ABB RAPID module: MainModule.mod

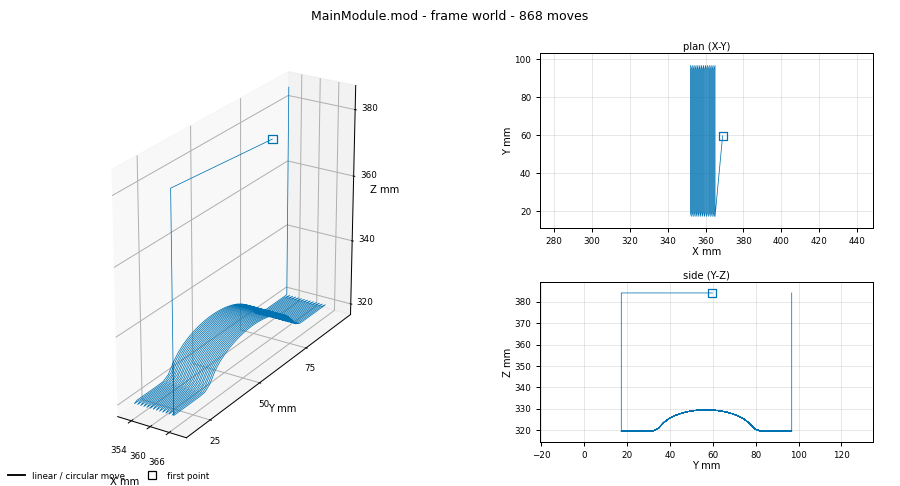
[picture p0: tool path of MainModule.mod in frame world, 868 of 868 moves have a stored position in this frame; points joined in program order, loops and branches not executed]
MODULE MainModule
PERS wobjdata Workobject_1:=[FALSE,TRUE,"",[[349,99.8,314.1],[0.707106781,0,0,-0.707106781]],[[0,0,0],[1,0,0,0]]];
PERS tooldata Extruder:=[TRUE,[[-32.5,-6.5,85.6],[0,-0.707106781,0.707106781,0]],[0.5,[-3,-15,42],[1,0,0,0],0,0,0]];
CONST robtarget p1 := [ [0,0,0], [1, 0, 0, 0], [0,0,0,0], [9E9,9E9, 9E9, 9E9, 9E9, 9E9] ];
VAR speeddata vel1 := [20,20,10,10];
VAR zonedata zoneval:=[FALSE,5,30,30,10,10,10];



PROC main()
AccSet 10,10;
SingArea\Wrist;
ConfL\On;

MoveL RelTool (p1,40.000000,20.000000,70.00000,\Rx:=0.000000,\Ry:=0.000000),vel1,z0,Extruder\WObj:=Workobject_1;
MoveL RelTool (p1,82.500000,16.000000,70.00000,\Rx:=0.000000,\Ry:=0.000000),vel1,z0,Extruder\WObj:=Workobject_1;


MoveL RelTool (p1,82.500000,16.000000,5.500000,\Rx:=0.000000,\Ry:=-0.000000),vel1,zoneval,Extruder\WObj:=Workobject_1;
MoveL RelTool (p1,80.000000,16.000000,5.500000,\Rx:=0.000000,\Ry:=-0.000000),vel1,zoneval,Extruder\WObj:=Workobject_1;
MoveL RelTool (p1,77.500000,16.000000,5.500000,\Rx:=0.000000,\Ry:=-0.000000),vel1,zoneval,Extruder\WObj:=Workobject_1;
MoveL RelTool (p1,75.000000,16.000000,5.500000,\Rx:=0.000000,\Ry:=-0.000000),vel1,zoneval,Extruder\WObj:=Workobject_1;
MoveL RelTool (p1,72.500000,16.000000,5.500000,\Rx:=0.000000,\Ry:=-0.000000),vel1,zoneval,Extruder\WObj:=Workobject_1;
MoveL RelTool (p1,70.000000,16.000000,5.500000,\Rx:=0.000000,\Ry:=-0.000000),vel1,zoneval,Extruder\WObj:=Workobject_1;
MoveL RelTool (p1,67.500000,16.000000,5.696103,\Rx:=0.000000,\Ry:=2.996421),vel1,zoneval,Extruder\WObj:=Workobject_1;
MoveL RelTool (p1,65.000000,16.000000,7.002928,\Rx:=0.000000,\Ry:=8.615508),vel1,zoneval,Extruder\WObj:=Workobject_1;
MoveL RelTool (p1,62.500000,16.000000,9.740509,\Rx:=0.000000,\Ry:=9.749555),vel1,zoneval,Extruder\WObj:=Workobject_1;
MoveL RelTool (p1,60.000000,16.000000,11.535030,\Rx:=0.000000,\Ry:=7.277441),vel1,zoneval,Extruder\WObj:=Workobject_1;
MoveL RelTool (p1,57.500000,16.000000,12.769306,\Rx:=0.000000,\Ry:=4.894735),vel1,zoneval,Extruder\WObj:=Workobject_1;
MoveL RelTool (p1,55.000000,16.000000,13.693467,\Rx:=0.000000,\Ry:=3.765598),vel1,zoneval,Extruder\WObj:=Workobject_1;
MoveL RelTool (p1,52.500000,16.000000,14.391107,\Rx:=0.000000,\Ry:=2.777529),vel1,zoneval,Extruder\WObj:=Workobject_1;
MoveL RelTool (p1,50.000000,16.000000,14.902666,\Rx:=0.000000,\Ry:=1.838961),vel1,zoneval,Extruder\WObj:=Workobject_1;
MoveL RelTool (p1,47.500000,16.000000,15.253646,\Rx:=0.000000,\Ry:=1.522915),vel1,zoneval,Extruder\WObj:=Workobject_1;
MoveL RelTool (p1,45.000000,16.000000,15.441995,\Rx:=0.000000,\Ry:=0.957446),vel1,zoneval,Extruder\WObj:=Workobject_1;
MoveL RelTool (p1,42.500000,16.000000,15.493202,\Rx:=0.000000,\Ry:=0.175753),vel1,zoneval,Extruder\WObj:=Workobject_1;
MoveL RelTool (p1,40.000000,16.000000,15.385044,\Rx:=0.000000,\Ry:=-0.609665),vel1,zoneval,Extruder\WObj:=Workobject_1;
MoveL RelTool (p1,37.500000,16.000000,15.140411,\Rx:=0.000000,\Ry:=-1.473255),vel1,zoneval,Extruder\WObj:=Workobject_1;
MoveL RelTool (p1,35.000000,16.000000,14.745289,\Rx:=0.000000,\Ry:=-2.361471),vel1,zoneval,Extruder\WObj:=Workobject_1;
MoveL RelTool (p1,32.500000,16.000000,14.177969,\Rx:=0.000000,\Ry:=-3.310711),vel1,zoneval,Extruder\WObj:=Workobject_1;
MoveL RelTool (p1,30.000000,16.000000,13.409588,\Rx:=0.000000,\Ry:=-4.304408),vel1,zoneval,Extruder\WObj:=Workobject_1;
MoveL RelTool (p1,27.500000,16.000000,12.393895,\Rx:=0.000000,\Ry:=-5.366573),vel1,zoneval,Extruder\WObj:=Workobject_1;
MoveL RelTool (p1,25.000000,16.000000,11.015814,\Rx:=0.000000,\Ry:=-7.116071),vel1,zoneval,Extruder\WObj:=Workobject_1;
MoveL RelTool (p1,22.500000,16.000000,8.916208,\Rx:=0.000000,\Ry:=-10.083054),vel1,zoneval,Extruder\WObj:=Workobject_1;
MoveL RelTool (p1,20.000000,16.000000,6.390765,\Rx:=0.000000,\Ry:=-7.195088),vel1,zoneval,Extruder\WObj:=Workobject_1;
MoveL RelTool (p1,17.500000,16.000000,5.549338,\Rx:=0.000000,\Ry:=-1.638714),vel1,zoneval,Extruder\WObj:=Workobject_1;
MoveL RelTool (p1,15.000000,16.000000,5.500000,\Rx:=0.000000,\Ry:=-0.000000),vel1,zoneval,Extruder\WObj:=Workobject_1;
MoveL RelTool (p1,12.500000,16.000000,5.500000,\Rx:=0.000000,\Ry:=-0.000000),vel1,zoneval,Extruder\WObj:=Workobject_1;
MoveL RelTool (p1,10.000000,16.000000,5.500000,\Rx:=0.000000,\Ry:=-0.000000),vel1,zoneval,Extruder\WObj:=Workobject_1;
MoveL RelTool (p1,7.500000,16.000000,5.500000,\Rx:=0.000000,\Ry:=-0.000000),vel1,zoneval,Extruder\WObj:=Workobject_1;
MoveL RelTool (p1,5.000000,16.000000,5.500000,\Rx:=0.000000,\Ry:=-0.000000),vel1,zoneval,Extruder\WObj:=Workobject_1;
MoveL RelTool (p1,3.000000,16.000000,5.500000,\Rx:=0.000000,\Ry:=0),vel1,zoneval,Extruder\WObj:=Workobject_1;
MoveL RelTool (p1,5.000000,15.500000,5.500000,\Rx:=0.000000,\Ry:=0.000000),vel1,zoneval,Extruder\WObj:=Workobject_1;
MoveL RelTool (p1,7.500000,15.500000,5.500000,\Rx:=0.000000,\Ry:=0.000000),vel1,zoneval,Extruder\WObj:=Workobject_1;
MoveL RelTool (p1,10.000000,15.500000,5.500000,\Rx:=0.000000,\Ry:=0.000000),vel1,zoneval,Extruder\WObj:=Workobject_1;
MoveL RelTool (p1,12.500000,15.500000,5.500000,\Rx:=0.000000,\Ry:=0.000000),vel1,zoneval,Extruder\WObj:=Workobject_1;
MoveL RelTool (p1,15.000000,15.500000,5.500000,\Rx:=0.000000,\Ry:=0.000000),vel1,zoneval,Extruder\WObj:=Workobject_1;
MoveL RelTool (p1,17.500000,15.500000,5.549338,\Rx:=0.000000,\Ry:=-1.027233),vel1,zoneval,Extruder\WObj:=Workobject_1;
MoveL RelTool (p1,20.000000,15.500000,6.390765,\Rx:=0.000000,\Ry:=-6.482955),vel1,zoneval,Extruder\WObj:=Workobject_1;
MoveL RelTool (p1,22.500000,15.500000,8.916208,\Rx:=0.000000,\Ry:=-11.282192),vel1,zoneval,Extruder\WObj:=Workobject_1;
MoveL RelTool (p1,25.000000,15.500000,11.015814,\Rx:=0.000000,\Ry:=-7.926142),vel1,zoneval,Extruder\WObj:=Workobject_1;
MoveL RelTool (p1,27.500000,15.500000,12.393895,\Rx:=0.000000,\Ry:=-5.366573),vel1,zoneval,Extruder\WObj:=Workobject_1;
MoveL RelTool (p1,30.000000,15.500000,13.409588,\Rx:=0.000000,\Ry:=-4.304408),vel1,zoneval,Extruder\WObj:=Workobject_1;
MoveL RelTool (p1,32.500000,15.500000,14.177969,\Rx:=0.000000,\Ry:=-3.310711),vel1,zoneval,Extruder\WObj:=Workobject_1;
MoveL RelTool (p1,35.000000,15.500000,14.745289,\Rx:=0.000000,\Ry:=-2.361471),vel1,zoneval,Extruder\WObj:=Workobject_1;
MoveL RelTool (p1,37.500000,15.500000,15.140411,\Rx:=0.000000,\Ry:=-1.473255),vel1,zoneval,Extruder\WObj:=Workobject_1;
MoveL RelTool (p1,40.000000,15.500000,15.385044,\Rx:=0.000000,\Ry:=-0.609665),vel1,zoneval,Extruder\WObj:=Workobject_1;
MoveL RelTool (p1,42.500000,15.500000,15.493202,\Rx:=0.000000,\Ry:=-0.313643),vel1,zoneval,Extruder\WObj:=Workobject_1;
MoveL RelTool (p1,45.000000,15.500000,15.441995,\Rx:=0.000000,\Ry:=0.600478),vel1,zoneval,Extruder\WObj:=Workobject_1;
MoveL RelTool (p1,47.500000,15.500000,15.253646,\Rx:=0.000000,\Ry:=0.957446),vel1,zoneval,Extruder\WObj:=Workobject_1;
MoveL RelTool (p1,50.000000,15.500000,14.902666,\Rx:=0.000000,\Ry:=1.838961),vel1,zoneval,Extruder\WObj:=Workobject_1;
MoveL RelTool (p1,52.500000,15.500000,14.391107,\Rx:=0.000000,\Ry:=2.777529),vel1,zoneval,Extruder\WObj:=Workobject_1;
MoveL RelTool (p1,55.000000,15.500000,13.693467,\Rx:=0.000000,\Ry:=3.765598),vel1,zoneval,Extruder\WObj:=Workobject_1;
MoveL RelTool (p1,57.500000,15.500000,12.769306,\Rx:=0.000000,\Ry:=4.809648),vel1,zoneval,Extruder\WObj:=Workobject_1;
MoveL RelTool (p1,60.000000,15.500000,11.535030,\Rx:=0.000000,\Ry:=6.353659),vel1,zoneval,Extruder\WObj:=Workobject_1;
MoveL RelTool (p1,62.500000,15.500000,9.740509,\Rx:=0.000000,\Ry:=8.756273),vel1,zoneval,Extruder\WObj:=Workobject_1;
MoveL RelTool (p1,65.000000,15.500000,7.002928,\Rx:=0.000000,\Ry:=9.759467),vel1,zoneval,Extruder\WObj:=Workobject_1;
MoveL RelTool (p1,67.500000,15.500000,5.696103,\Rx:=0.000000,\Ry:=3.252694),vel1,zoneval,Extruder\WObj:=Workobject_1;
MoveL RelTool (p1,70.000000,15.500000,5.500000,\Rx:=0.000000,\Ry:=0.000000),vel1,zoneval,Extruder\WObj:=Workobject_1;
MoveL RelTool (p1,72.500000,15.500000,5.500000,\Rx:=0.000000,\Ry:=0.000000),vel1,zoneval,Extruder\WObj:=Workobject_1;
MoveL RelTool (p1,75.000000,15.500000,5.500000,\Rx:=0.000000,\Ry:=0.000000),vel1,zoneval,Extruder\WObj:=Workobject_1;
MoveL RelTool (p1,77.500000,15.500000,5.500000,\Rx:=0.000000,\Ry:=0.000000),vel1,zoneval,Extruder\WObj:=Workobject_1;
MoveL RelTool (p1,80.000000,15.500000,5.500000,\Rx:=0.000000,\Ry:=0.000000),vel1,zoneval,Extruder\WObj:=Workobject_1;
MoveL RelTool (p1,82.500000,15.500000,5.500000,\Rx:=0.000000,\Ry:=0.000000),vel1,zoneval,Extruder\WObj:=Workobject_1;
MoveL RelTool (p1,80.500000,15.000000,5.500000,\Rx:=0.000000,\Ry:=-0.000000),vel1,zoneval,Extruder\WObj:=Workobject_1;
MoveL RelTool (p1,78.000000,15.000000,5.500000,\Rx:=0.000000,\Ry:=-0.000000),vel1,zoneval,Extruder\WObj:=Workobject_1;
MoveL RelTool (p1,75.500000,15.000000,5.500000,\Rx:=0.000000,\Ry:=-0.000000),vel1,zoneval,Extruder\WObj:=Workobject_1;
MoveL RelTool (p1,73.000000,15.000000,5.500000,\Rx:=0.000000,\Ry:=-0.000000),vel1,zoneval,Extruder\WObj:=Workobject_1;
MoveL RelTool (p1,70.500000,15.000000,5.500000,\Rx:=0.000000,\Ry:=-0.000000),vel1,zoneval,Extruder\WObj:=Workobject_1;
MoveL RelTool (p1,68.000000,15.000000,5.576212,\Rx:=0.000000,\Ry:=1.027235),vel1,zoneval,Extruder\WObj:=Workobject_1;
MoveL RelTool (p1,65.500000,15.000000,6.601352,\Rx:=0.000000,\Ry:=7.190651),vel1,zoneval,Extruder\WObj:=Workobject_1;
MoveL RelTool (p1,63.000000,15.000000,9.259802,\Rx:=0.000000,\Ry:=10.438096),vel1,zoneval,Extruder\WObj:=Workobject_1;
MoveL RelTool (p1,60.500000,15.000000,11.213438,\Rx:=0.000000,\Ry:=7.277441),vel1,zoneval,Extruder\WObj:=Workobject_1;
MoveL RelTool (p1,58.000000,15.000000,12.567025,\Rx:=0.000000,\Ry:=5.967579),vel1,zoneval,Extruder\WObj:=Workobject_1;
MoveL RelTool (p1,55.500000,15.000000,13.541124,\Rx:=0.000000,\Ry:=4.323199),vel1,zoneval,Extruder\WObj:=Workobject_1;
MoveL RelTool (p1,53.000000,15.000000,14.280270,\Rx:=0.000000,\Ry:=3.233363),vel1,zoneval,Extruder\WObj:=Workobject_1;
MoveL RelTool (p1,50.500000,15.000000,14.829944,\Rx:=0.000000,\Ry:=2.667808),vel1,zoneval,Extruder\WObj:=Workobject_1;
MoveL RelTool (p1,48.000000,15.000000,15.193555,\Rx:=0.000000,\Ry:=1.838961),vel1,zoneval,Extruder\WObj:=Workobject_1;
MoveL RelTool (p1,45.500000,15.000000,15.404325,\Rx:=0.000000,\Ry:=0.957446),vel1,zoneval,Extruder\WObj:=Workobject_1;
MoveL RelTool (p1,43.000000,15.000000,15.486300,\Rx:=0.000000,\Ry:=0.175753),vel1,zoneval,Extruder\WObj:=Workobject_1;
MoveL RelTool (p1,40.500000,15.000000,15.409004,\Rx:=0.000000,\Ry:=-0.609665),vel1,zoneval,Extruder\WObj:=Workobject_1;
MoveL RelTool (p1,38.000000,15.000000,15.198525,\Rx:=0.000000,\Ry:=-1.473255),vel1,zoneval,Extruder\WObj:=Workobject_1;
MoveL RelTool (p1,35.500000,15.000000,14.839102,\Rx:=0.000000,\Ry:=-2.361471),vel1,zoneval,Extruder\WObj:=Workobject_1;
MoveL RelTool (p1,33.000000,15.000000,14.310992,\Rx:=0.000000,\Ry:=-3.310711),vel1,zoneval,Extruder\WObj:=Workobject_1;
MoveL RelTool (p1,30.500000,15.000000,13.585370,\Rx:=0.000000,\Ry:=-4.304408),vel1,zoneval,Extruder\WObj:=Workobject_1;
MoveL RelTool (p1,28.000000,15.000000,12.618075,\Rx:=0.000000,\Ry:=-5.366573),vel1,zoneval,Extruder\WObj:=Workobject_1;
MoveL RelTool (p1,25.500000,15.000000,11.328519,\Rx:=0.000000,\Ry:=-6.568275),vel1,zoneval,Extruder\WObj:=Workobject_1;
MoveL RelTool (p1,23.000000,15.000000,9.422774,\Rx:=0.000000,\Ry:=-9.481583),vel1,zoneval,Extruder\WObj:=Workobject_1;
MoveL RelTool (p1,20.500000,15.000000,6.707804,\Rx:=0.000000,\Ry:=-9.245066),vel1,zoneval,Extruder\WObj:=Workobject_1;
MoveL RelTool (p1,18.000000,15.000000,5.614048,\Rx:=0.000000,\Ry:=-3.081691),vel1,zoneval,Extruder\WObj:=Workobject_1;
MoveL RelTool (p1,15.500000,15.000000,5.500000,\Rx:=0.000000,\Ry:=-0.000000),vel1,zoneval,Extruder\WObj:=Workobject_1;
MoveL RelTool (p1,13.000000,15.000000,5.500000,\Rx:=0.000000,\Ry:=-0.000000),vel1,zoneval,Extruder\WObj:=Workobject_1;
MoveL RelTool (p1,10.500000,15.000000,5.500000,\Rx:=0.000000,\Ry:=-0.000000),vel1,zoneval,Extruder\WObj:=Workobject_1;
MoveL RelTool (p1,8.000000,15.000000,5.500000,\Rx:=0.000000,\Ry:=-0.000000),vel1,zoneval,Extruder\WObj:=Workobject_1;
MoveL RelTool (p1,5.500000,15.000000,5.500000,\Rx:=0.000000,\Ry:=-0.000000),vel1,zoneval,Extruder\WObj:=Workobject_1;
MoveL RelTool (p1,3.000000,15.000000,5.500000,\Rx:=0.000000,\Ry:=-0.000000),vel1,zoneval,Extruder\WObj:=Workobject_1;
MoveL RelTool (p1,5.000000,14.500000,5.500000,\Rx:=0.000000,\Ry:=0.000000),vel1,zoneval,Extruder\WObj:=Workobject_1;
MoveL RelTool (p1,7.500000,14.500000,5.500000,\Rx:=0.000000,\Ry:=0.000000),vel1,zoneval,Extruder\WObj:=Workobject_1;
MoveL RelTool (p1,10.000000,14.500000,5.500000,\Rx:=0.000000,\Ry:=0.000000),vel1,zoneval,Extruder\WObj:=Workobject_1;
MoveL RelTool (p1,12.500000,14.500000,5.500000,\Rx:=0.000000,\Ry:=0.000000),vel1,zoneval,Extruder\WObj:=Workobject_1;
MoveL RelTool (p1,15.000000,14.500000,5.500000,\Rx:=0.000000,\Ry:=0.000000),vel1,zoneval,Extruder\WObj:=Workobject_1;
MoveL RelTool (p1,17.500000,14.500000,5.549338,\Rx:=0.000000,\Ry:=-1.027233),vel1,zoneval,Extruder\WObj:=Workobject_1;
MoveL RelTool (p1,20.000000,14.500000,6.390765,\Rx:=0.000000,\Ry:=-6.482955),vel1,zoneval,Extruder\WObj:=Workobject_1;
MoveL RelTool (p1,22.500000,14.500000,8.916208,\Rx:=0.000000,\Ry:=-11.282192),vel1,zoneval,Extruder\WObj:=Workobject_1;
MoveL RelTool (p1,25.000000,14.500000,11.015814,\Rx:=0.000000,\Ry:=-7.926142),vel1,zoneval,Extruder\WObj:=Workobject_1;
MoveL RelTool (p1,27.500000,14.500000,12.393895,\Rx:=0.000000,\Ry:=-5.366573),vel1,zoneval,Extruder\WObj:=Workobject_1;
MoveL RelTool (p1,30.000000,14.500000,13.409588,\Rx:=0.000000,\Ry:=-4.304408),vel1,zoneval,Extruder\WObj:=Workobject_1;
MoveL RelTool (p1,32.500000,14.500000,14.177969,\Rx:=0.000000,\Ry:=-3.310711),vel1,zoneval,Extruder\WObj:=Workobject_1;
MoveL RelTool (p1,35.000000,14.500000,14.745289,\Rx:=0.000000,\Ry:=-2.361471),vel1,zoneval,Extruder\WObj:=Workobject_1;
MoveL RelTool (p1,37.500000,14.500000,15.140411,\Rx:=0.000000,\Ry:=-1.473255),vel1,zoneval,Extruder\WObj:=Workobject_1;
MoveL RelTool (p1,40.000000,14.500000,15.385044,\Rx:=0.000000,\Ry:=-0.609665),vel1,zoneval,Extruder\WObj:=Workobject_1;
MoveL RelTool (p1,42.500000,14.500000,15.493202,\Rx:=0.000000,\Ry:=-0.313643),vel1,zoneval,Extruder\WObj:=Workobject_1;
MoveL RelTool (p1,45.000000,14.500000,15.441995,\Rx:=0.000000,\Ry:=0.600478),vel1,zoneval,Extruder\WObj:=Workobject_1;
MoveL RelTool (p1,47.500000,14.500000,15.253646,\Rx:=0.000000,\Ry:=0.957446),vel1,zoneval,Extruder\WObj:=Workobject_1;
MoveL RelTool (p1,50.000000,14.500000,14.902666,\Rx:=0.000000,\Ry:=1.838961),vel1,zoneval,Extruder\WObj:=Workobject_1;
MoveL RelTool (p1,52.500000,14.500000,14.391107,\Rx:=0.000000,\Ry:=2.777529),vel1,zoneval,Extruder\WObj:=Workobject_1;
MoveL RelTool (p1,55.000000,14.500000,13.693467,\Rx:=0.000000,\Ry:=3.765598),vel1,zoneval,Extruder\WObj:=Workobject_1;
MoveL RelTool (p1,57.500000,14.500000,12.769306,\Rx:=0.000000,\Ry:=4.809648),vel1,zoneval,Extruder\WObj:=Workobject_1;
MoveL RelTool (p1,60.000000,14.500000,11.535030,\Rx:=0.000000,\Ry:=6.353659),vel1,zoneval,Extruder\WObj:=Workobject_1;
MoveL RelTool (p1,62.500000,14.500000,9.740509,\Rx:=0.000000,\Ry:=8.756273),vel1,zoneval,Extruder\WObj:=Workobject_1;
MoveL RelTool (p1,65.000000,14.500000,7.002928,\Rx:=0.000000,\Ry:=9.759467),vel1,zoneval,Extruder\WObj:=Workobject_1;
MoveL RelTool (p1,67.500000,14.500000,5.696103,\Rx:=0.000000,\Ry:=3.252694),vel1,zoneval,Extruder\WObj:=Workobject_1;
MoveL RelTool (p1,70.000000,14.500000,5.500000,\Rx:=0.000000,\Ry:=0.000000),vel1,zoneval,Extruder\WObj:=Workobject_1;
MoveL RelTool (p1,72.500000,14.500000,5.500000,\Rx:=0.000000,\Ry:=0.000000),vel1,zoneval,Extruder\WObj:=Workobject_1;
MoveL RelTool (p1,75.000000,14.500000,5.500000,\Rx:=0.000000,\Ry:=0.000000),vel1,zoneval,Extruder\WObj:=Workobject_1;
MoveL RelTool (p1,77.500000,14.500000,5.500000,\Rx:=0.000000,\Ry:=0.000000),vel1,zoneval,Extruder\WObj:=Workobject_1;
MoveL RelTool (p1,80.000000,14.500000,5.500000,\Rx:=0.000000,\Ry:=0.000000),vel1,zoneval,Extruder\WObj:=Workobject_1;
MoveL RelTool (p1,82.500000,14.500000,5.500000,\Rx:=0.000000,\Ry:=0.000000),vel1,zoneval,Extruder\WObj:=Workobject_1;
MoveL RelTool (p1,80.500000,14.000000,5.500000,\Rx:=0.000000,\Ry:=-0.000000),vel1,zoneval,Extruder\WObj:=Workobject_1;
MoveL RelTool (p1,78.000000,14.000000,5.500000,\Rx:=0.000000,\Ry:=-0.000000),vel1,zoneval,Extruder\WObj:=Workobject_1;
MoveL RelTool (p1,75.500000,14.000000,5.500000,\Rx:=0.000000,\Ry:=-0.000000),vel1,zoneval,Extruder\WObj:=Workobject_1;
MoveL RelTool (p1,73.000000,14.000000,5.500000,\Rx:=0.000000,\Ry:=-0.000000),vel1,zoneval,Extruder\WObj:=Workobject_1;
MoveL RelTool (p1,70.500000,14.000000,5.500000,\Rx:=0.000000,\Ry:=-0.000000),vel1,zoneval,Extruder\WObj:=Workobject_1;
MoveL RelTool (p1,68.000000,14.000000,5.576212,\Rx:=0.000000,\Ry:=1.027235),vel1,zoneval,Extruder\WObj:=Workobject_1;
MoveL RelTool (p1,65.500000,14.000000,6.601352,\Rx:=0.000000,\Ry:=7.190651),vel1,zoneval,Extruder\WObj:=Workobject_1;
MoveL RelTool (p1,63.000000,14.000000,9.259802,\Rx:=0.000000,\Ry:=10.438096),vel1,zoneval,Extruder\WObj:=Workobject_1;
MoveL RelTool (p1,60.500000,14.000000,11.213438,\Rx:=0.000000,\Ry:=7.277441),vel1,zoneval,Extruder\WObj:=Workobject_1;
MoveL RelTool (p1,58.000000,14.000000,12.567025,\Rx:=0.000000,\Ry:=5.967579),vel1,zoneval,Extruder\WObj:=Workobject_1;
MoveL RelTool (p1,55.500000,14.000000,13.541124,\Rx:=0.000000,\Ry:=4.323199),vel1,zoneval,Extruder\WObj:=Workobject_1;
MoveL RelTool (p1,53.000000,14.000000,14.280270,\Rx:=0.000000,\Ry:=3.233363),vel1,zoneval,Extruder\WObj:=Workobject_1;
MoveL RelTool (p1,50.500000,14.000000,14.829944,\Rx:=0.000000,\Ry:=2.667808),vel1,zoneval,Extruder\WObj:=Workobject_1;
MoveL RelTool (p1,48.000000,14.000000,15.193555,\Rx:=0.000000,\Ry:=1.838961),vel1,zoneval,Extruder\WObj:=Workobject_1;
MoveL RelTool (p1,45.500000,14.000000,15.404325,\Rx:=0.000000,\Ry:=0.957446),vel1,zoneval,Extruder\WObj:=Workobject_1;
MoveL RelTool (p1,43.000000,14.000000,15.486300,\Rx:=0.000000,\Ry:=0.175753),vel1,zoneval,Extruder\WObj:=Workobject_1;
MoveL RelTool (p1,40.500000,14.000000,15.409004,\Rx:=0.000000,\Ry:=-0.609665),vel1,zoneval,Extruder\WObj:=Workobject_1;
MoveL RelTool (p1,38.000000,14.000000,15.198525,\Rx:=0.000000,\Ry:=-1.473255),vel1,zoneval,Extruder\WObj:=Workobject_1;
MoveL RelTool (p1,35.500000,14.000000,14.839102,\Rx:=0.000000,\Ry:=-2.361471),vel1,zoneval,Extruder\WObj:=Workobject_1;
MoveL RelTool (p1,33.000000,14.000000,14.310992,\Rx:=0.000000,\Ry:=-3.310711),vel1,zoneval,Extruder\WObj:=Workobject_1;
MoveL RelTool (p1,30.500000,14.000000,13.585370,\Rx:=0.000000,\Ry:=-4.304408),vel1,zoneval,Extruder\WObj:=Workobject_1;
MoveL RelTool (p1,28.000000,14.000000,12.618075,\Rx:=0.000000,\Ry:=-5.366573),vel1,zoneval,Extruder\WObj:=Workobject_1;
MoveL RelTool (p1,25.500000,14.000000,11.328519,\Rx:=0.000000,\Ry:=-6.568275),vel1,zoneval,Extruder\WObj:=Workobject_1;
MoveL RelTool (p1,23.000000,14.000000,9.422774,\Rx:=0.000000,\Ry:=-9.481583),vel1,zoneval,Extruder\WObj:=Workobject_1;
MoveL RelTool (p1,20.500000,14.000000,6.707804,\Rx:=0.000000,\Ry:=-9.245066),vel1,zoneval,Extruder\WObj:=Workobject_1;
MoveL RelTool (p1,18.000000,14.000000,5.614048,\Rx:=0.000000,\Ry:=-3.081691),vel1,zoneval,Extruder\WObj:=Workobject_1;
MoveL RelTool (p1,15.500000,14.000000,5.500000,\Rx:=0.000000,\Ry:=-0.000000),vel1,zoneval,Extruder\WObj:=Workobject_1;
MoveL RelTool (p1,13.000000,14.000000,5.500000,\Rx:=0.000000,\Ry:=-0.000000),vel1,zoneval,Extruder\WObj:=Workobject_1;
MoveL RelTool (p1,10.500000,14.000000,5.500000,\Rx:=0.000000,\Ry:=-0.000000),vel1,zoneval,Extruder\WObj:=Workobject_1;
MoveL RelTool (p1,8.000000,14.000000,5.500000,\Rx:=0.000000,\Ry:=-0.000000),vel1,zoneval,Extruder\WObj:=Workobject_1;
MoveL RelTool (p1,5.500000,14.000000,5.500000,\Rx:=0.000000,\Ry:=-0.000000),vel1,zoneval,Extruder\WObj:=Workobject_1;
MoveL RelTool (p1,3.000000,14.000000,5.500000,\Rx:=0.000000,\Ry:=-0.000000),vel1,zoneval,Extruder\WObj:=Workobject_1;
MoveL RelTool (p1,5.000000,13.500000,5.500000,\Rx:=0.000000,\Ry:=0.000000),vel1,zoneval,Extruder\WObj:=Workobject_1;
MoveL RelTool (p1,7.500000,13.500000,5.500000,\Rx:=0.000000,\Ry:=0.000000),vel1,zoneval,Extruder\WObj:=Workobject_1;
MoveL RelTool (p1,10.000000,13.500000,5.500000,\Rx:=0.000000,\Ry:=0.000000),vel1,zoneval,Extruder\WObj:=Workobject_1;
MoveL RelTool (p1,12.500000,13.500000,5.500000,\Rx:=0.000000,\Ry:=0.000000),vel1,zoneval,Extruder\WObj:=Workobject_1;
MoveL RelTool (p1,15.000000,13.500000,5.500000,\Rx:=0.000000,\Ry:=0.000000),vel1,zoneval,Extruder\WObj:=Workobject_1;
MoveL RelTool (p1,17.500000,13.500000,5.549338,\Rx:=0.000000,\Ry:=-1.027233),vel1,zoneval,Extruder\WObj:=Workobject_1;
MoveL RelTool (p1,20.000000,13.500000,6.390765,\Rx:=0.000000,\Ry:=-6.482955),vel1,zoneval,Extruder\WObj:=Workobject_1;
MoveL RelTool (p1,22.500000,13.500000,8.916208,\Rx:=0.000000,\Ry:=-11.282192),vel1,zoneval,Extruder\WObj:=Workobject_1;
MoveL RelTool (p1,25.000000,13.500000,11.015814,\Rx:=0.000000,\Ry:=-7.926142),vel1,zoneval,Extruder\WObj:=Workobject_1;
MoveL RelTool (p1,27.500000,13.500000,12.393895,\Rx:=0.000000,\Ry:=-5.366573),vel1,zoneval,Extruder\WObj:=Workobject_1;
MoveL RelTool (p1,30.000000,13.500000,13.409588,\Rx:=0.000000,\Ry:=-4.304408),vel1,zoneval,Extruder\WObj:=Workobject_1;
MoveL RelTool (p1,32.500000,13.500000,14.177969,\Rx:=0.000000,\Ry:=-3.310711),vel1,zoneval,Extruder\WObj:=Workobject_1;
MoveL RelTool (p1,35.000000,13.500000,14.745289,\Rx:=0.000000,\Ry:=-2.361471),vel1,zoneval,Extruder\WObj:=Workobject_1;
MoveL RelTool (p1,37.500000,13.500000,15.140411,\Rx:=0.000000,\Ry:=-1.473255),vel1,zoneval,Extruder\WObj:=Workobject_1;
MoveL RelTool (p1,40.000000,13.500000,15.385044,\Rx:=0.000000,\Ry:=-0.609665),vel1,zoneval,Extruder\WObj:=Workobject_1;
MoveL RelTool (p1,42.500000,13.500000,15.493202,\Rx:=0.000000,\Ry:=-0.313643),vel1,zoneval,Extruder\WObj:=Workobject_1;
MoveL RelTool (p1,45.000000,13.500000,15.441995,\Rx:=0.000000,\Ry:=0.600478),vel1,zoneval,Extruder\WObj:=Workobject_1;
MoveL RelTool (p1,47.500000,13.500000,15.253646,\Rx:=0.000000,\Ry:=0.957446),vel1,zoneval,Extruder\WObj:=Workobject_1;
MoveL RelTool (p1,50.000000,13.500000,14.902666,\Rx:=0.000000,\Ry:=1.838961),vel1,zoneval,Extruder\WObj:=Workobject_1;
MoveL RelTool (p1,52.500000,13.500000,14.391107,\Rx:=0.000000,\Ry:=2.777529),vel1,zoneval,Extruder\WObj:=Workobject_1;
MoveL RelTool (p1,55.000000,13.500000,13.693467,\Rx:=0.000000,\Ry:=3.765598),vel1,zoneval,Extruder\WObj:=Workobject_1;
MoveL RelTool (p1,57.500000,13.500000,12.769306,\Rx:=0.000000,\Ry:=4.809648),vel1,zoneval,Extruder\WObj:=Workobject_1;
MoveL RelTool (p1,60.000000,13.500000,11.535030,\Rx:=0.000000,\Ry:=6.353659),vel1,zoneval,Extruder\WObj:=Workobject_1;
MoveL RelTool (p1,62.500000,13.500000,9.740509,\Rx:=0.000000,\Ry:=8.756273),vel1,zoneval,Extruder\WObj:=Workobject_1;
MoveL RelTool (p1,65.000000,13.500000,7.002928,\Rx:=0.000000,\Ry:=9.759467),vel1,zoneval,Extruder\WObj:=Workobject_1;
MoveL RelTool (p1,67.500000,13.500000,5.696103,\Rx:=0.000000,\Ry:=3.252694),vel1,zoneval,Extruder\WObj:=Workobject_1;
MoveL RelTool (p1,70.000000,13.500000,5.500000,\Rx:=0.000000,\Ry:=0.000000),vel1,zoneval,Extruder\WObj:=Workobject_1;
MoveL RelTool (p1,72.500000,13.500000,5.500000,\Rx:=0.000000,\Ry:=0.000000),vel1,zoneval,Extruder\WObj:=Workobject_1;
MoveL RelTool (p1,75.000000,13.500000,5.500000,\Rx:=0.000000,\Ry:=0.000000),vel1,zoneval,Extruder\WObj:=Workobject_1;
MoveL RelTool (p1,77.500000,13.500000,5.500000,\Rx:=0.000000,\Ry:=0.000000),vel1,zoneval,Extruder\WObj:=Workobject_1;
MoveL RelTool (p1,80.000000,13.500000,5.500000,\Rx:=0.000000,\Ry:=0.000000),vel1,zoneval,Extruder\WObj:=Workobject_1;
MoveL RelTool (p1,82.500000,13.500000,5.500000,\Rx:=0.000000,\Ry:=0.000000),vel1,zoneval,Extruder\WObj:=Workobject_1;
MoveL RelTool (p1,80.500000,13.000000,5.500000,\Rx:=0.000000,\Ry:=-0.000000),vel1,zoneval,Extruder\WObj:=Workobject_1;
MoveL RelTool (p1,78.000000,13.000000,5.500000,\Rx:=0.000000,\Ry:=-0.000000),vel1,zoneval,Extruder\WObj:=Workobject_1;
MoveL RelTool (p1,75.500000,13.000000,5.500000,\Rx:=0.000000,\Ry:=-0.000000),vel1,zoneval,Extruder\WObj:=Workobject_1;
MoveL RelTool (p1,73.000000,13.000000,5.500000,\Rx:=0.000000,\Ry:=-0.000000),vel1,zoneval,Extruder\WObj:=Workobject_1;
MoveL RelTool (p1,70.500000,13.000000,5.500000,\Rx:=0.000000,\Ry:=-0.000000),vel1,zoneval,Extruder\WObj:=Workobject_1;
MoveL RelTool (p1,68.000000,13.000000,5.576212,\Rx:=0.000000,\Ry:=1.027235),vel1,zoneval,Extruder\WObj:=Workobject_1;
MoveL RelTool (p1,65.500000,13.000000,6.601352,\Rx:=0.000000,\Ry:=7.190651),vel1,zoneval,Extruder\WObj:=Workobject_1;
MoveL RelTool (p1,63.000000,13.000000,9.259802,\Rx:=0.000000,\Ry:=10.438096),vel1,zoneval,Extruder\WObj:=Workobject_1;
MoveL RelTool (p1,60.500000,13.000000,11.213438,\Rx:=0.000000,\Ry:=7.277441),vel1,zoneval,Extruder\WObj:=Workobject_1;
MoveL RelTool (p1,58.000000,13.000000,12.567025,\Rx:=0.000000,\Ry:=5.967579),vel1,zoneval,Extruder\WObj:=Workobject_1;
MoveL RelTool (p1,55.500000,13.000000,13.541124,\Rx:=0.000000,\Ry:=4.323199),vel1,zoneval,Extruder\WObj:=Workobject_1;
MoveL RelTool (p1,53.000000,13.000000,14.280270,\Rx:=0.000000,\Ry:=3.233363),vel1,zoneval,Extruder\WObj:=Workobject_1;
MoveL RelTool (p1,50.500000,13.000000,14.829944,\Rx:=0.000000,\Ry:=2.667808),vel1,zoneval,Extruder\WObj:=Workobject_1;
MoveL RelTool (p1,48.000000,13.000000,15.193555,\Rx:=0.000000,\Ry:=1.838961),vel1,zoneval,Extruder\WObj:=Workobject_1;
MoveL RelTool (p1,45.500000,13.000000,15.404325,\Rx:=0.000000,\Ry:=0.957446),vel1,zoneval,Extruder\WObj:=Workobject_1;
MoveL RelTool (p1,43.000000,13.000000,15.486300,\Rx:=0.000000,\Ry:=0.175753),vel1,zoneval,Extruder\WObj:=Workobject_1;
MoveL RelTool (p1,40.500000,13.000000,15.409004,\Rx:=0.000000,\Ry:=-0.609665),vel1,zoneval,Extruder\WObj:=Workobject_1;
MoveL RelTool (p1,38.000000,13.000000,15.198525,\Rx:=0.000000,\Ry:=-1.473255),vel1,zoneval,Extruder\WObj:=Workobject_1;
MoveL RelTool (p1,35.500000,13.000000,14.839102,\Rx:=0.000000,\Ry:=-2.361471),vel1,zoneval,Extruder\WObj:=Workobject_1;
MoveL RelTool (p1,33.000000,13.000000,14.310992,\Rx:=0.000000,\Ry:=-3.310711),vel1,zoneval,Extruder\WObj:=Workobject_1;
MoveL RelTool (p1,30.500000,13.000000,13.585370,\Rx:=0.000000,\Ry:=-4.304408),vel1,zoneval,Extruder\WObj:=Workobject_1;
MoveL RelTool (p1,28.000000,13.000000,12.618075,\Rx:=0.000000,\Ry:=-5.366573),vel1,zoneval,Extruder\WObj:=Workobject_1;
MoveL RelTool (p1,25.500000,13.000000,11.328519,\Rx:=0.000000,\Ry:=-6.568275),vel1,zoneval,Extruder\WObj:=Workobject_1;
MoveL RelTool (p1,23.000000,13.000000,9.422774,\Rx:=0.000000,\Ry:=-9.481583),vel1,zoneval,Extruder\WObj:=Workobject_1;
MoveL RelTool (p1,20.500000,13.000000,6.707804,\Rx:=0.000000,\Ry:=-9.245066),vel1,zoneval,Extruder\WObj:=Workobject_1;
MoveL RelTool (p1,18.000000,13.000000,5.614048,\Rx:=0.000000,\Ry:=-3.081691),vel1,zoneval,Extruder\WObj:=Workobject_1;
MoveL RelTool (p1,15.500000,13.000000,5.500000,\Rx:=0.000000,\Ry:=-0.000000),vel1,zoneval,Extruder\WObj:=Workobject_1;
MoveL RelTool (p1,13.000000,13.000000,5.500000,\Rx:=0.000000,\Ry:=-0.000000),vel1,zoneval,Extruder\WObj:=Workobject_1;
MoveL RelTool (p1,10.500000,13.000000,5.500000,\Rx:=0.000000,\Ry:=-0.000000),vel1,zoneval,Extruder\WObj:=Workobject_1;
MoveL RelTool (p1,8.000000,13.000000,5.500000,\Rx:=0.000000,\Ry:=-0.000000),vel1,zoneval,Extruder\WObj:=Workobject_1;
MoveL RelTool (p1,5.500000,13.000000,5.500000,\Rx:=0.000000,\Ry:=-0.000000),vel1,zoneval,Extruder\WObj:=Workobject_1;
MoveL RelTool (p1,3.000000,13.000000,5.500000,\Rx:=0.000000,\Ry:=-0.000000),vel1,zoneval,Extruder\WObj:=Workobject_1;
MoveL RelTool (p1,5.000000,12.500000,5.500000,\Rx:=0.000000,\Ry:=0.000000),vel1,zoneval,Extruder\WObj:=Workobject_1;
MoveL RelTool (p1,7.500000,12.500000,5.500000,\Rx:=0.000000,\Ry:=0.000000),vel1,zoneval,Extruder\WObj:=Workobject_1;
MoveL RelTool (p1,10.000000,12.500000,5.500000,\Rx:=0.000000,\Ry:=0.000000),vel1,zoneval,Extruder\WObj:=Workobject_1;
MoveL RelTool (p1,12.500000,12.500000,5.500000,\Rx:=0.000000,\Ry:=0.000000),vel1,zoneval,Extruder\WObj:=Workobject_1;
MoveL RelTool (p1,15.000000,12.500000,5.500000,\Rx:=0.000000,\Ry:=0.000000),vel1,zoneval,Extruder\WObj:=Workobject_1;
MoveL RelTool (p1,17.500000,12.500000,5.549338,\Rx:=0.000000,\Ry:=-1.027233),vel1,zoneval,Extruder\WObj:=Workobject_1;
MoveL RelTool (p1,20.000000,12.500000,6.390765,\Rx:=0.000000,\Ry:=-6.482955),vel1,zoneval,Extruder\WObj:=Workobject_1;
MoveL RelTool (p1,22.500000,12.500000,8.916208,\Rx:=0.000000,\Ry:=-11.282192),vel1,zoneval,Extruder\WObj:=Workobject_1;
MoveL RelTool (p1,25.000000,12.500000,11.015814,\Rx:=0.000000,\Ry:=-7.926142),vel1,zoneval,Extruder\WObj:=Workobject_1;
MoveL RelTool (p1,27.500000,12.500000,12.393895,\Rx:=0.000000,\Ry:=-5.366573),vel1,zoneval,Extruder\WObj:=Workobject_1;
MoveL RelTool (p1,30.000000,12.500000,13.409588,\Rx:=0.000000,\Ry:=-4.304408),vel1,zoneval,Extruder\WObj:=Workobject_1;
MoveL RelTool (p1,32.500000,12.500000,14.177969,\Rx:=0.000000,\Ry:=-3.310711),vel1,zoneval,Extruder\WObj:=Workobject_1;
MoveL RelTool (p1,35.000000,12.500000,14.745289,\Rx:=0.000000,\Ry:=-2.361471),vel1,zoneval,Extruder\WObj:=Workobject_1;
MoveL RelTool (p1,37.500000,12.500000,15.140411,\Rx:=0.000000,\Ry:=-1.473255),vel1,zoneval,Extruder\WObj:=Workobject_1;
MoveL RelTool (p1,40.000000,12.500000,15.385044,\Rx:=0.000000,\Ry:=-0.609665),vel1,zoneval,Extruder\WObj:=Workobject_1;
MoveL RelTool (p1,42.500000,12.500000,15.493202,\Rx:=0.000000,\Ry:=-0.313643),vel1,zoneval,Extruder\WObj:=Workobject_1;
MoveL RelTool (p1,45.000000,12.500000,15.441995,\Rx:=0.000000,\Ry:=0.600478),vel1,zoneval,Extruder\WObj:=Workobject_1;
MoveL RelTool (p1,47.500000,12.500000,15.253646,\Rx:=0.000000,\Ry:=0.957446),vel1,zoneval,Extruder\WObj:=Workobject_1;
MoveL RelTool (p1,50.000000,12.500000,14.902666,\Rx:=0.000000,\Ry:=1.838961),vel1,zoneval,Extruder\WObj:=Workobject_1;
MoveL RelTool (p1,52.500000,12.500000,14.391107,\Rx:=0.000000,\Ry:=2.777529),vel1,zoneval,Extruder\WObj:=Workobject_1;
MoveL RelTool (p1,55.000000,12.500000,13.693467,\Rx:=0.000000,\Ry:=3.765598),vel1,zoneval,Extruder\WObj:=Workobject_1;
MoveL RelTool (p1,57.500000,12.500000,12.769306,\Rx:=0.000000,\Ry:=4.809648),vel1,zoneval,Extruder\WObj:=Workobject_1;
MoveL RelTool (p1,60.000000,12.500000,11.535030,\Rx:=0.000000,\Ry:=6.353659),vel1,zoneval,Extruder\WObj:=Workobject_1;
MoveL RelTool (p1,62.500000,12.500000,9.740509,\Rx:=0.000000,\Ry:=8.756273),vel1,zoneval,Extruder\WObj:=Workobject_1;
MoveL RelTool (p1,65.000000,12.500000,7.002928,\Rx:=0.000000,\Ry:=9.759467),vel1,zoneval,Extruder\WObj:=Workobject_1;
MoveL RelTool (p1,67.500000,12.500000,5.696103,\Rx:=0.000000,\Ry:=3.252694),vel1,zoneval,Extruder\WObj:=Workobject_1;
MoveL RelTool (p1,70.000000,12.500000,5.500000,\Rx:=0.000000,\Ry:=0.000000),vel1,zoneval,Extruder\WObj:=Workobject_1;
MoveL RelTool (p1,72.500000,12.500000,5.500000,\Rx:=0.000000,\Ry:=0.000000),vel1,zoneval,Extruder\WObj:=Workobject_1;
MoveL RelTool (p1,75.000000,12.500000,5.500000,\Rx:=0.000000,\Ry:=0.000000),vel1,zoneval,Extruder\WObj:=Workobject_1;
MoveL RelTool (p1,77.500000,12.500000,5.500000,\Rx:=0.000000,\Ry:=0.000000),vel1,zoneval,Extruder\WObj:=Workobject_1;
MoveL RelTool (p1,80.000000,12.500000,5.500000,\Rx:=0.000000,\Ry:=0.000000),vel1,zoneval,Extruder\WObj:=Workobject_1;
MoveL RelTool (p1,82.500000,12.500000,5.500000,\Rx:=0.000000,\Ry:=0.000000),vel1,zoneval,Extruder\WObj:=Workobject_1;
MoveL RelTool (p1,80.500000,12.000000,5.500000,\Rx:=0.000000,\Ry:=-0.000000),vel1,zoneval,Extruder\WObj:=Workobject_1;
MoveL RelTool (p1,78.000000,12.000000,5.500000,\Rx:=0.000000,\Ry:=-0.000000),vel1,zoneval,Extruder\WObj:=Workobject_1;
MoveL RelTool (p1,75.500000,12.000000,5.500000,\Rx:=0.000000,\Ry:=-0.000000),vel1,zoneval,Extruder\WObj:=Workobject_1;
MoveL RelTool (p1,73.000000,12.000000,5.500000,\Rx:=0.000000,\Ry:=-0.000000),vel1,zoneval,Extruder\WObj:=Workobject_1;
MoveL RelTool (p1,70.500000,12.000000,5.500000,\Rx:=0.000000,\Ry:=-0.000000),vel1,zoneval,Extruder\WObj:=Workobject_1;
MoveL RelTool (p1,68.000000,12.000000,5.576212,\Rx:=0.000000,\Ry:=1.027235),vel1,zoneval,Extruder\WObj:=Workobject_1;
MoveL RelTool (p1,65.500000,12.000000,6.601352,\Rx:=0.000000,\Ry:=7.190651),vel1,zoneval,Extruder\WObj:=Workobject_1;
MoveL RelTool (p1,63.000000,12.000000,9.259802,\Rx:=0.000000,\Ry:=10.438096),vel1,zoneval,Extruder\WObj:=Workobject_1;
MoveL RelTool (p1,60.500000,12.000000,11.213438,\Rx:=0.000000,\Ry:=7.277441),vel1,zoneval,Extruder\WObj:=Workobject_1;
MoveL RelTool (p1,58.000000,12.000000,12.567025,\Rx:=0.000000,\Ry:=5.967579),vel1,zoneval,Extruder\WObj:=Workobject_1;
MoveL RelTool (p1,55.500000,12.000000,13.541124,\Rx:=0.000000,\Ry:=4.323199),vel1,zoneval,Extruder\WObj:=Workobject_1;
MoveL RelTool (p1,53.000000,12.000000,14.280270,\Rx:=0.000000,\Ry:=3.233363),vel1,zoneval,Extruder\WObj:=Workobject_1;
MoveL RelTool (p1,50.500000,12.000000,14.829944,\Rx:=0.000000,\Ry:=2.667808),vel1,zoneval,Extruder\WObj:=Workobject_1;
MoveL RelTool (p1,48.000000,12.000000,15.193555,\Rx:=0.000000,\Ry:=1.838961),vel1,zoneval,Extruder\WObj:=Workobject_1;
MoveL RelTool (p1,45.500000,12.000000,15.404325,\Rx:=0.000000,\Ry:=0.957446),vel1,zoneval,Extruder\WObj:=Workobject_1;
MoveL RelTool (p1,43.000000,12.000000,15.486300,\Rx:=0.000000,\Ry:=0.175753),vel1,zoneval,Extruder\WObj:=Workobject_1;
MoveL RelTool (p1,40.500000,12.000000,15.409004,\Rx:=0.000000,\Ry:=-0.609665),vel1,zoneval,Extruder\WObj:=Workobject_1;
MoveL RelTool (p1,38.000000,12.000000,15.198525,\Rx:=0.000000,\Ry:=-1.473255),vel1,zoneval,Extruder\WObj:=Workobject_1;
MoveL RelTool (p1,35.500000,12.000000,14.839102,\Rx:=0.000000,\Ry:=-2.361471),vel1,zoneval,Extruder\WObj:=Workobject_1;
MoveL RelTool (p1,33.000000,12.000000,14.310992,\Rx:=0.000000,\Ry:=-3.310711),vel1,zoneval,Extruder\WObj:=Workobject_1;
MoveL RelTool (p1,30.500000,12.000000,13.585370,\Rx:=0.000000,\Ry:=-4.304408),vel1,zoneval,Extruder\WObj:=Workobject_1;
MoveL RelTool (p1,28.000000,12.000000,12.618075,\Rx:=0.000000,\Ry:=-5.366573),vel1,zoneval,Extruder\WObj:=Workobject_1;
MoveL RelTool (p1,25.500000,12.000000,11.328519,\Rx:=0.000000,\Ry:=-6.568275),vel1,zoneval,Extruder\WObj:=Workobject_1;
MoveL RelTool (p1,23.000000,12.000000,9.422774,\Rx:=0.000000,\Ry:=-9.481583),vel1,zoneval,Extruder\WObj:=Workobject_1;
MoveL RelTool (p1,20.500000,12.000000,6.707804,\Rx:=0.000000,\Ry:=-9.245066),vel1,zoneval,Extruder\WObj:=Workobject_1;
MoveL RelTool (p1,18.000000,12.000000,5.614048,\Rx:=0.000000,\Ry:=-3.081691),vel1,zoneval,Extruder\WObj:=Workobject_1;
MoveL RelTool (p1,15.500000,12.000000,5.500000,\Rx:=0.000000,\Ry:=-0.000000),vel1,zoneval,Extruder\WObj:=Workobject_1;
MoveL RelTool (p1,13.000000,12.000000,5.500000,\Rx:=0.000000,\Ry:=-0.000000),vel1,zoneval,Extruder\WObj:=Workobject_1;
MoveL RelTool (p1,10.500000,12.000000,5.500000,\Rx:=0.000000,\Ry:=-0.000000),vel1,zoneval,Extruder\WObj:=Workobject_1;
MoveL RelTool (p1,8.000000,12.000000,5.500000,\Rx:=0.000000,\Ry:=-0.000000),vel1,zoneval,Extruder\WObj:=Workobject_1;
MoveL RelTool (p1,5.500000,12.000000,5.500000,\Rx:=0.000000,\Ry:=-0.000000),vel1,zoneval,Extruder\WObj:=Workobject_1;
MoveL RelTool (p1,3.000000,12.000000,5.500000,\Rx:=0.000000,\Ry:=-0.000000),vel1,zoneval,Extruder\WObj:=Workobject_1;
MoveL RelTool (p1,5.000000,11.500000,5.500000,\Rx:=0.000000,\Ry:=0.000000),vel1,zoneval,Extruder\WObj:=Workobject_1;
MoveL RelTool (p1,7.500000,11.500000,5.500000,\Rx:=0.000000,\Ry:=0.000000),vel1,zoneval,Extruder\WObj:=Workobject_1;
MoveL RelTool (p1,10.000000,11.500000,5.500000,\Rx:=0.000000,\Ry:=0.000000),vel1,zoneval,Extruder\WObj:=Workobject_1;
MoveL RelTool (p1,12.500000,11.500000,5.500000,\Rx:=0.000000,\Ry:=0.000000),vel1,zoneval,Extruder\WObj:=Workobject_1;
MoveL RelTool (p1,15.000000,11.500000,5.500000,\Rx:=0.000000,\Ry:=0.000000),vel1,zoneval,Extruder\WObj:=Workobject_1;
MoveL RelTool (p1,17.500000,11.500000,5.549338,\Rx:=0.000000,\Ry:=-1.027233),vel1,zoneval,Extruder\WObj:=Workobject_1;
MoveL RelTool (p1,20.000000,11.500000,6.390765,\Rx:=0.000000,\Ry:=-6.482955),vel1,zoneval,Extruder\WObj:=Workobject_1;
MoveL RelTool (p1,22.500000,11.500000,8.916208,\Rx:=0.000000,\Ry:=-11.282192),vel1,zoneval,Extruder\WObj:=Workobject_1;
MoveL RelTool (p1,25.000000,11.500000,11.015814,\Rx:=0.000000,\Ry:=-7.926142),vel1,zoneval,Extruder\WObj:=Workobject_1;
MoveL RelTool (p1,27.500000,11.500000,12.393895,\Rx:=0.000000,\Ry:=-5.366573),vel1,zoneval,Extruder\WObj:=Workobject_1;
MoveL RelTool (p1,30.000000,11.500000,13.409588,\Rx:=0.000000,\Ry:=-4.304408),vel1,zoneval,Extruder\WObj:=Workobject_1;
MoveL RelTool (p1,32.500000,11.500000,14.177969,\Rx:=0.000000,\Ry:=-3.310711),vel1,zoneval,Extruder\WObj:=Workobject_1;
MoveL RelTool (p1,35.000000,11.500000,14.745289,\Rx:=0.000000,\Ry:=-2.361471),vel1,zoneval,Extruder\WObj:=Workobject_1;
MoveL RelTool (p1,37.500000,11.500000,15.140411,\Rx:=0.000000,\Ry:=-1.473255),vel1,zoneval,Extruder\WObj:=Workobject_1;
MoveL RelTool (p1,40.000000,11.500000,15.385044,\Rx:=0.000000,\Ry:=-0.609665),vel1,zoneval,Extruder\WObj:=Workobject_1;
MoveL RelTool (p1,42.500000,11.500000,15.493202,\Rx:=0.000000,\Ry:=-0.313643),vel1,zoneval,Extruder\WObj:=Workobject_1;
MoveL RelTool (p1,45.000000,11.500000,15.441995,\Rx:=0.000000,\Ry:=0.600478),vel1,zoneval,Extruder\WObj:=Workobject_1;
MoveL RelTool (p1,47.500000,11.500000,15.253646,\Rx:=0.000000,\Ry:=0.957446),vel1,zoneval,Extruder\WObj:=Workobject_1;
MoveL RelTool (p1,50.000000,11.500000,14.902666,\Rx:=0.000000,\Ry:=1.838961),vel1,zoneval,Extruder\WObj:=Workobject_1;
MoveL RelTool (p1,52.500000,11.500000,14.391107,\Rx:=0.000000,\Ry:=2.777529),vel1,zoneval,Extruder\WObj:=Workobject_1;
MoveL RelTool (p1,55.000000,11.500000,13.693467,\Rx:=0.000000,\Ry:=3.765598),vel1,zoneval,Extruder\WObj:=Workobject_1;
MoveL RelTool (p1,57.500000,11.500000,12.769306,\Rx:=0.000000,\Ry:=4.809648),vel1,zoneval,Extruder\WObj:=Workobject_1;
MoveL RelTool (p1,60.000000,11.500000,11.535030,\Rx:=0.000000,\Ry:=6.353659),vel1,zoneval,Extruder\WObj:=Workobject_1;
MoveL RelTool (p1,62.500000,11.500000,9.740509,\Rx:=0.000000,\Ry:=8.756273),vel1,zoneval,Extruder\WObj:=Workobject_1;
MoveL RelTool (p1,65.000000,11.500000,7.002928,\Rx:=0.000000,\Ry:=9.759467),vel1,zoneval,Extruder\WObj:=Workobject_1;
MoveL RelTool (p1,67.500000,11.500000,5.696103,\Rx:=0.000000,\Ry:=3.252694),vel1,zoneval,Extruder\WObj:=Workobject_1;
MoveL RelTool (p1,70.000000,11.500000,5.500000,\Rx:=0.000000,\Ry:=0.000000),vel1,zoneval,Extruder\WObj:=Workobject_1;
MoveL RelTool (p1,72.500000,11.500000,5.500000,\Rx:=0.000000,\Ry:=0.000000),vel1,zoneval,Extruder\WObj:=Workobject_1;
MoveL RelTool (p1,75.000000,11.500000,5.500000,\Rx:=0.000000,\Ry:=0.000000),vel1,zoneval,Extruder\WObj:=Workobject_1;
MoveL RelTool (p1,77.500000,11.500000,5.500000,\Rx:=0.000000,\Ry:=0.000000),vel1,zoneval,Extruder\WObj:=Workobject_1;
MoveL RelTool (p1,80.000000,11.500000,5.500000,\Rx:=0.000000,\Ry:=0.000000),vel1,zoneval,Extruder\WObj:=Workobject_1;
MoveL RelTool (p1,82.500000,11.500000,5.500000,\Rx:=0.000000,\Ry:=0.000000),vel1,zoneval,Extruder\WObj:=Workobject_1;
MoveL RelTool (p1,80.500000,11.000000,5.500000,\Rx:=0.000000,\Ry:=-0.000000),vel1,zoneval,Extruder\WObj:=Workobject_1;
MoveL RelTool (p1,78.000000,11.000000,5.500000,\Rx:=0.000000,\Ry:=-0.000000),vel1,zoneval,Extruder\WObj:=Workobject_1;
MoveL RelTool (p1,75.500000,11.000000,5.500000,\Rx:=0.000000,\Ry:=-0.000000),vel1,zoneval,Extruder\WObj:=Workobject_1;
MoveL RelTool (p1,73.000000,11.000000,5.500000,\Rx:=0.000000,\Ry:=-0.000000),vel1,zoneval,Extruder\WObj:=Workobject_1;
MoveL RelTool (p1,70.500000,11.000000,5.500000,\Rx:=0.000000,\Ry:=-0.000000),vel1,zoneval,Extruder\WObj:=Workobject_1;
MoveL RelTool (p1,68.000000,11.000000,5.576212,\Rx:=0.000000,\Ry:=1.027235),vel1,zoneval,Extruder\WObj:=Workobject_1;
MoveL RelTool (p1,65.500000,11.000000,6.601352,\Rx:=0.000000,\Ry:=7.190651),vel1,zoneval,Extruder\WObj:=Workobject_1;
MoveL RelTool (p1,63.000000,11.000000,9.259802,\Rx:=0.000000,\Ry:=10.438096),vel1,zoneval,Extruder\WObj:=Workobject_1;
MoveL RelTool (p1,60.500000,11.000000,11.213438,\Rx:=0.000000,\Ry:=7.277441),vel1,zoneval,Extruder\WObj:=Workobject_1;
MoveL RelTool (p1,58.000000,11.000000,12.567025,\Rx:=0.000000,\Ry:=5.967579),vel1,zoneval,Extruder\WObj:=Workobject_1;
MoveL RelTool (p1,55.500000,11.000000,13.541124,\Rx:=0.000000,\Ry:=4.323199),vel1,zoneval,Extruder\WObj:=Workobject_1;
MoveL RelTool (p1,53.000000,11.000000,14.280270,\Rx:=0.000000,\Ry:=3.233363),vel1,zoneval,Extruder\WObj:=Workobject_1;
MoveL RelTool (p1,50.500000,11.000000,14.829944,\Rx:=0.000000,\Ry:=2.667808),vel1,zoneval,Extruder\WObj:=Workobject_1;
MoveL RelTool (p1,48.000000,11.000000,15.193555,\Rx:=0.000000,\Ry:=1.838961),vel1,zoneval,Extruder\WObj:=Workobject_1;
MoveL RelTool (p1,45.500000,11.000000,15.404325,\Rx:=0.000000,\Ry:=0.957446),vel1,zoneval,Extruder\WObj:=Workobject_1;
MoveL RelTool (p1,43.000000,11.000000,15.486300,\Rx:=0.000000,\Ry:=0.175753),vel1,zoneval,Extruder\WObj:=Workobject_1;
MoveL RelTool (p1,40.500000,11.000000,15.409004,\Rx:=0.000000,\Ry:=-0.609665),vel1,zoneval,Extruder\WObj:=Workobject_1;
MoveL RelTool (p1,38.000000,11.000000,15.198525,\Rx:=0.000000,\Ry:=-1.473255),vel1,zoneval,Extruder\WObj:=Workobject_1;
MoveL RelTool (p1,35.500000,11.000000,14.839102,\Rx:=0.000000,\Ry:=-2.361471),vel1,zoneval,Extruder\WObj:=Workobject_1;
MoveL RelTool (p1,33.000000,11.000000,14.310992,\Rx:=0.000000,\Ry:=-3.310711),vel1,zoneval,Extruder\WObj:=Workobject_1;
MoveL RelTool (p1,30.500000,11.000000,13.585370,\Rx:=0.000000,\Ry:=-4.304408),vel1,zoneval,Extruder\WObj:=Workobject_1;
MoveL RelTool (p1,28.000000,11.000000,12.618075,\Rx:=0.000000,\Ry:=-5.366573),vel1,zoneval,Extruder\WObj:=Workobject_1;
MoveL RelTool (p1,25.500000,11.000000,11.328519,\Rx:=0.000000,\Ry:=-6.568275),vel1,zoneval,Extruder\WObj:=Workobject_1;
MoveL RelTool (p1,23.000000,11.000000,9.422774,\Rx:=0.000000,\Ry:=-9.481583),vel1,zoneval,Extruder\WObj:=Workobject_1;
MoveL RelTool (p1,20.500000,11.000000,6.707804,\Rx:=0.000000,\Ry:=-9.245066),vel1,zoneval,Extruder\WObj:=Workobject_1;
MoveL RelTool (p1,18.000000,11.000000,5.614048,\Rx:=0.000000,\Ry:=-3.081691),vel1,zoneval,Extruder\WObj:=Workobject_1;
MoveL RelTool (p1,15.500000,11.000000,5.500000,\Rx:=0.000000,\Ry:=-0.000000),vel1,zoneval,Extruder\WObj:=Workobject_1;
MoveL RelTool (p1,13.000000,11.000000,5.500000,\Rx:=0.000000,\Ry:=-0.000000),vel1,zoneval,Extruder\WObj:=Workobject_1;
MoveL RelTool (p1,10.500000,11.000000,5.500000,\Rx:=0.000000,\Ry:=-0.000000),vel1,zoneval,Extruder\WObj:=Workobject_1;
MoveL RelTool (p1,8.000000,11.000000,5.500000,\Rx:=0.000000,\Ry:=-0.000000),vel1,zoneval,Extruder\WObj:=Workobject_1;
MoveL RelTool (p1,5.500000,11.000000,5.500000,\Rx:=0.000000,\Ry:=-0.000000),vel1,zoneval,Extruder\WObj:=Workobject_1;
MoveL RelTool (p1,3.000000,11.000000,5.500000,\Rx:=0.000000,\Ry:=-0.000000),vel1,zoneval,Extruder\WObj:=Workobject_1;
MoveL RelTool (p1,5.000000,10.500000,5.500000,\Rx:=0.000000,\Ry:=0.000000),vel1,zoneval,Extruder\WObj:=Workobject_1;
MoveL RelTool (p1,7.500000,10.500000,5.500000,\Rx:=0.000000,\Ry:=0.000000),vel1,zoneval,Extruder\WObj:=Workobject_1;
MoveL RelTool (p1,10.000000,10.500000,5.500000,\Rx:=0.000000,\Ry:=0.000000),vel1,zoneval,Extruder\WObj:=Workobject_1;
MoveL RelTool (p1,12.500000,10.500000,5.500000,\Rx:=0.000000,\Ry:=0.000000),vel1,zoneval,Extruder\WObj:=Workobject_1;
MoveL RelTool (p1,15.000000,10.500000,5.500000,\Rx:=0.000000,\Ry:=0.000000),vel1,zoneval,Extruder\WObj:=Workobject_1;
MoveL RelTool (p1,17.500000,10.500000,5.549338,\Rx:=0.000000,\Ry:=-1.027233),vel1,zoneval,Extruder\WObj:=Workobject_1;
MoveL RelTool (p1,20.000000,10.500000,6.390765,\Rx:=0.000000,\Ry:=-6.482955),vel1,zoneval,Extruder\WObj:=Workobject_1;
MoveL RelTool (p1,22.500000,10.500000,8.916208,\Rx:=0.000000,\Ry:=-11.282192),vel1,zoneval,Extruder\WObj:=Workobject_1;
MoveL RelTool (p1,25.000000,10.500000,11.015814,\Rx:=0.000000,\Ry:=-7.926142),vel1,zoneval,Extruder\WObj:=Workobject_1;
MoveL RelTool (p1,27.500000,10.500000,12.393895,\Rx:=0.000000,\Ry:=-5.366573),vel1,zoneval,Extruder\WObj:=Workobject_1;
MoveL RelTool (p1,30.000000,10.500000,13.409588,\Rx:=0.000000,\Ry:=-4.304408),vel1,zoneval,Extruder\WObj:=Workobject_1;
MoveL RelTool (p1,32.500000,10.500000,14.177969,\Rx:=0.000000,\Ry:=-3.310711),vel1,zoneval,Extruder\WObj:=Workobject_1;
MoveL RelTool (p1,35.000000,10.500000,14.745289,\Rx:=0.000000,\Ry:=-2.361471),vel1,zoneval,Extruder\WObj:=Workobject_1;
MoveL RelTool (p1,37.500000,10.500000,15.140411,\Rx:=0.000000,\Ry:=-1.473255),vel1,zoneval,Extruder\WObj:=Workobject_1;
MoveL RelTool (p1,40.000000,10.500000,15.385044,\Rx:=0.000000,\Ry:=-0.609665),vel1,zoneval,Extruder\WObj:=Workobject_1;
MoveL RelTool (p1,42.500000,10.500000,15.493202,\Rx:=0.000000,\Ry:=-0.313643),vel1,zoneval,Extruder\WObj:=Workobject_1;
MoveL RelTool (p1,45.000000,10.500000,15.441995,\Rx:=0.000000,\Ry:=0.600478),vel1,zoneval,Extruder\WObj:=Workobject_1;
MoveL RelTool (p1,47.500000,10.500000,15.253646,\Rx:=0.000000,\Ry:=0.957446),vel1,zoneval,Extruder\WObj:=Workobject_1;
MoveL RelTool (p1,50.000000,10.500000,14.902666,\Rx:=0.000000,\Ry:=1.838961),vel1,zoneval,Extruder\WObj:=Workobject_1;
MoveL RelTool (p1,52.500000,10.500000,14.391107,\Rx:=0.000000,\Ry:=2.777529),vel1,zoneval,Extruder\WObj:=Workobject_1;
MoveL RelTool (p1,55.000000,10.500000,13.693467,\Rx:=0.000000,\Ry:=3.765598),vel1,zoneval,Extruder\WObj:=Workobject_1;
MoveL RelTool (p1,57.500000,10.500000,12.769306,\Rx:=0.000000,\Ry:=4.809648),vel1,zoneval,Extruder\WObj:=Workobject_1;
MoveL RelTool (p1,60.000000,10.500000,11.535030,\Rx:=0.000000,\Ry:=6.353659),vel1,zoneval,Extruder\WObj:=Workobject_1;
MoveL RelTool (p1,62.500000,10.500000,9.740509,\Rx:=0.000000,\Ry:=8.756273),vel1,zoneval,Extruder\WObj:=Workobject_1;
MoveL RelTool (p1,65.000000,10.500000,7.002928,\Rx:=0.000000,\Ry:=9.759467),vel1,zoneval,Extruder\WObj:=Workobject_1;
MoveL RelTool (p1,67.500000,10.500000,5.696103,\Rx:=0.000000,\Ry:=3.252694),vel1,zoneval,Extruder\WObj:=Workobject_1;
MoveL RelTool (p1,70.000000,10.500000,5.500000,\Rx:=0.000000,\Ry:=0.000000),vel1,zoneval,Extruder\WObj:=Workobject_1;
MoveL RelTool (p1,72.500000,10.500000,5.500000,\Rx:=0.000000,\Ry:=0.000000),vel1,zoneval,Extruder\WObj:=Workobject_1;
MoveL RelTool (p1,75.000000,10.500000,5.500000,\Rx:=0.000000,\Ry:=0.000000),vel1,zoneval,Extruder\WObj:=Workobject_1;
MoveL RelTool (p1,77.500000,10.500000,5.500000,\Rx:=0.000000,\Ry:=0.000000),vel1,zoneval,Extruder\WObj:=Workobject_1;
MoveL RelTool (p1,80.000000,10.500000,5.500000,\Rx:=0.000000,\Ry:=0.000000),vel1,zoneval,Extruder\WObj:=Workobject_1;
MoveL RelTool (p1,82.500000,10.500000,5.500000,\Rx:=0.000000,\Ry:=0.000000),vel1,zoneval,Extruder\WObj:=Workobject_1;
MoveL RelTool (p1,80.500000,10.000000,5.500000,\Rx:=0.000000,\Ry:=-0.000000),vel1,zoneval,Extruder\WObj:=Workobject_1;
MoveL RelTool (p1,78.000000,10.000000,5.500000,\Rx:=0.000000,\Ry:=-0.000000),vel1,zoneval,Extruder\WObj:=Workobject_1;
MoveL RelTool (p1,75.500000,10.000000,5.500000,\Rx:=0.000000,\Ry:=-0.000000),vel1,zoneval,Extruder\WObj:=Workobject_1;
MoveL RelTool (p1,73.000000,10.000000,5.500000,\Rx:=0.000000,\Ry:=-0.000000),vel1,zoneval,Extruder\WObj:=Workobject_1;
MoveL RelTool (p1,70.500000,10.000000,5.500000,\Rx:=0.000000,\Ry:=-0.000000),vel1,zoneval,Extruder\WObj:=Workobject_1;
MoveL RelTool (p1,68.000000,10.000000,5.576212,\Rx:=0.000000,\Ry:=1.027235),vel1,zoneval,Extruder\WObj:=Workobject_1;
MoveL RelTool (p1,65.500000,10.000000,6.601352,\Rx:=0.000000,\Ry:=7.190651),vel1,zoneval,Extruder\WObj:=Workobject_1;
MoveL RelTool (p1,63.000000,10.000000,9.259802,\Rx:=0.000000,\Ry:=10.438096),vel1,zoneval,Extruder\WObj:=Workobject_1;
MoveL RelTool (p1,60.500000,10.000000,11.213438,\Rx:=0.000000,\Ry:=7.277441),vel1,zoneval,Extruder\WObj:=Workobject_1;
MoveL RelTool (p1,58.000000,10.000000,12.567025,\Rx:=0.000000,\Ry:=5.967579),vel1,zoneval,Extruder\WObj:=Workobject_1;
MoveL RelTool (p1,55.500000,10.000000,13.541124,\Rx:=0.000000,\Ry:=4.323199),vel1,zoneval,Extruder\WObj:=Workobject_1;
MoveL RelTool (p1,53.000000,10.000000,14.280270,\Rx:=0.000000,\Ry:=3.233363),vel1,zoneval,Extruder\WObj:=Workobject_1;
MoveL RelTool (p1,50.500000,10.000000,14.829944,\Rx:=0.000000,\Ry:=2.667808),vel1,zoneval,Extruder\WObj:=Workobject_1;
MoveL RelTool (p1,48.000000,10.000000,15.193555,\Rx:=0.000000,\Ry:=1.838961),vel1,zoneval,Extruder\WObj:=Workobject_1;
MoveL RelTool (p1,45.500000,10.000000,15.404325,\Rx:=0.000000,\Ry:=0.957446),vel1,zoneval,Extruder\WObj:=Workobject_1;
MoveL RelTool (p1,43.000000,10.000000,15.486300,\Rx:=0.000000,\Ry:=0.175753),vel1,zoneval,Extruder\WObj:=Workobject_1;
MoveL RelTool (p1,40.500000,10.000000,15.409004,\Rx:=0.000000,\Ry:=-0.609665),vel1,zoneval,Extruder\WObj:=Workobject_1;
MoveL RelTool (p1,38.000000,10.000000,15.198525,\Rx:=0.000000,\Ry:=-1.473255),vel1,zoneval,Extruder\WObj:=Workobject_1;
MoveL RelTool (p1,35.500000,10.000000,14.839102,\Rx:=0.000000,\Ry:=-2.361471),vel1,zoneval,Extruder\WObj:=Workobject_1;
MoveL RelTool (p1,33.000000,10.000000,14.310992,\Rx:=0.000000,\Ry:=-3.310711),vel1,zoneval,Extruder\WObj:=Workobject_1;
MoveL RelTool (p1,30.500000,10.000000,13.585370,\Rx:=0.000000,\Ry:=-4.304408),vel1,zoneval,Extruder\WObj:=Workobject_1;
MoveL RelTool (p1,28.000000,10.000000,12.618075,\Rx:=0.000000,\Ry:=-5.366573),vel1,zoneval,Extruder\WObj:=Workobject_1;
MoveL RelTool (p1,25.500000,10.000000,11.328519,\Rx:=0.000000,\Ry:=-6.568275),vel1,zoneval,Extruder\WObj:=Workobject_1;
MoveL RelTool (p1,23.000000,10.000000,9.422774,\Rx:=0.000000,\Ry:=-9.481583),vel1,zoneval,Extruder\WObj:=Workobject_1;
MoveL RelTool (p1,20.500000,10.000000,6.707804,\Rx:=0.000000,\Ry:=-9.245066),vel1,zoneval,Extruder\WObj:=Workobject_1;
MoveL RelTool (p1,18.000000,10.000000,5.614048,\Rx:=0.000000,\Ry:=-3.081691),vel1,zoneval,Extruder\WObj:=Workobject_1;
MoveL RelTool (p1,15.500000,10.000000,5.500000,\Rx:=0.000000,\Ry:=-0.000000),vel1,zoneval,Extruder\WObj:=Workobject_1;
MoveL RelTool (p1,13.000000,10.000000,5.500000,\Rx:=0.000000,\Ry:=-0.000000),vel1,zoneval,Extruder\WObj:=Workobject_1;
MoveL RelTool (p1,10.500000,10.000000,5.500000,\Rx:=0.000000,\Ry:=-0.000000),vel1,zoneval,Extruder\WObj:=Workobject_1;
MoveL RelTool (p1,8.000000,10.000000,5.500000,\Rx:=0.000000,\Ry:=-0.000000),vel1,zoneval,Extruder\WObj:=Workobject_1;
MoveL RelTool (p1,5.500000,10.000000,5.500000,\Rx:=0.000000,\Ry:=-0.000000),vel1,zoneval,Extruder\WObj:=Workobject_1;
MoveL RelTool (p1,3.000000,10.000000,5.500000,\Rx:=0.000000,\Ry:=-0.000000),vel1,zoneval,Extruder\WObj:=Workobject_1;
MoveL RelTool (p1,5.000000,9.500000,5.500000,\Rx:=0.000000,\Ry:=0.000000),vel1,zoneval,Extruder\WObj:=Workobject_1;
MoveL RelTool (p1,7.500000,9.500000,5.500000,\Rx:=0.000000,\Ry:=0.000000),vel1,zoneval,Extruder\WObj:=Workobject_1;
MoveL RelTool (p1,10.000000,9.500000,5.500000,\Rx:=0.000000,\Ry:=0.000000),vel1,zoneval,Extruder\WObj:=Workobject_1;
MoveL RelTool (p1,12.500000,9.500000,5.500000,\Rx:=0.000000,\Ry:=0.000000),vel1,zoneval,Extruder\WObj:=Workobject_1;
MoveL RelTool (p1,15.000000,9.500000,5.500000,\Rx:=0.000000,\Ry:=0.000000),vel1,zoneval,Extruder\WObj:=Workobject_1;
MoveL RelTool (p1,17.500000,9.500000,5.549338,\Rx:=0.000000,\Ry:=-1.027233),vel1,zoneval,Extruder\WObj:=Workobject_1;
MoveL RelTool (p1,20.000000,9.500000,6.390765,\Rx:=0.000000,\Ry:=-6.482955),vel1,zoneval,Extruder\WObj:=Workobject_1;
MoveL RelTool (p1,22.500000,9.500000,8.916208,\Rx:=0.000000,\Ry:=-11.282192),vel1,zoneval,Extruder\WObj:=Workobject_1;
MoveL RelTool (p1,25.000000,9.500000,11.015814,\Rx:=0.000000,\Ry:=-7.926142),vel1,zoneval,Extruder\WObj:=Workobject_1;
MoveL RelTool (p1,27.500000,9.500000,12.393895,\Rx:=0.000000,\Ry:=-5.366573),vel1,zoneval,Extruder\WObj:=Workobject_1;
MoveL RelTool (p1,30.000000,9.500000,13.409588,\Rx:=0.000000,\Ry:=-4.304408),vel1,zoneval,Extruder\WObj:=Workobject_1;
MoveL RelTool (p1,32.500000,9.500000,14.177969,\Rx:=0.000000,\Ry:=-3.310711),vel1,zoneval,Extruder\WObj:=Workobject_1;
MoveL RelTool (p1,35.000000,9.500000,14.745289,\Rx:=0.000000,\Ry:=-2.361471),vel1,zoneval,Extruder\WObj:=Workobject_1;
MoveL RelTool (p1,37.500000,9.500000,15.140411,\Rx:=0.000000,\Ry:=-1.473255),vel1,zoneval,Extruder\WObj:=Workobject_1;
MoveL RelTool (p1,40.000000,9.500000,15.385044,\Rx:=0.000000,\Ry:=-0.609665),vel1,zoneval,Extruder\WObj:=Workobject_1;
MoveL RelTool (p1,42.500000,9.500000,15.493202,\Rx:=0.000000,\Ry:=-0.313643),vel1,zoneval,Extruder\WObj:=Workobject_1;
MoveL RelTool (p1,45.000000,9.500000,15.441995,\Rx:=0.000000,\Ry:=0.600478),vel1,zoneval,Extruder\WObj:=Workobject_1;
MoveL RelTool (p1,47.500000,9.500000,15.253646,\Rx:=0.000000,\Ry:=0.957446),vel1,zoneval,Extruder\WObj:=Workobject_1;
MoveL RelTool (p1,50.000000,9.500000,14.902666,\Rx:=0.000000,\Ry:=1.838961),vel1,zoneval,Extruder\WObj:=Workobject_1;
MoveL RelTool (p1,52.500000,9.500000,14.391107,\Rx:=0.000000,\Ry:=2.777529),vel1,zoneval,Extruder\WObj:=Workobject_1;
MoveL RelTool (p1,55.000000,9.500000,13.693467,\Rx:=0.000000,\Ry:=3.765598),vel1,zoneval,Extruder\WObj:=Workobject_1;
MoveL RelTool (p1,57.500000,9.500000,12.769306,\Rx:=0.000000,\Ry:=4.809648),vel1,zoneval,Extruder\WObj:=Workobject_1;
MoveL RelTool (p1,60.000000,9.500000,11.535030,\Rx:=0.000000,\Ry:=6.353659),vel1,zoneval,Extruder\WObj:=Workobject_1;
MoveL RelTool (p1,62.500000,9.500000,9.740509,\Rx:=0.000000,\Ry:=8.756273),vel1,zoneval,Extruder\WObj:=Workobject_1;
MoveL RelTool (p1,65.000000,9.500000,7.002928,\Rx:=0.000000,\Ry:=9.759467),vel1,zoneval,Extruder\WObj:=Workobject_1;
MoveL RelTool (p1,67.500000,9.500000,5.696103,\Rx:=0.000000,\Ry:=3.252694),vel1,zoneval,Extruder\WObj:=Workobject_1;
MoveL RelTool (p1,70.000000,9.500000,5.500000,\Rx:=0.000000,\Ry:=0.000000),vel1,zoneval,Extruder\WObj:=Workobject_1;
MoveL RelTool (p1,72.500000,9.500000,5.500000,\Rx:=0.000000,\Ry:=0.000000),vel1,zoneval,Extruder\WObj:=Workobject_1;
MoveL RelTool (p1,75.000000,9.500000,5.500000,\Rx:=0.000000,\Ry:=0.000000),vel1,zoneval,Extruder\WObj:=Workobject_1;
MoveL RelTool (p1,77.500000,9.500000,5.500000,\Rx:=0.000000,\Ry:=0.000000),vel1,zoneval,Extruder\WObj:=Workobject_1;
MoveL RelTool (p1,80.000000,9.500000,5.500000,\Rx:=0.000000,\Ry:=0.000000),vel1,zoneval,Extruder\WObj:=Workobject_1;
MoveL RelTool (p1,82.500000,9.500000,5.500000,\Rx:=0.000000,\Ry:=0.000000),vel1,zoneval,Extruder\WObj:=Workobject_1;
MoveL RelTool (p1,80.500000,9.000000,5.500000,\Rx:=0.000000,\Ry:=-0.000000),vel1,zoneval,Extruder\WObj:=Workobject_1;
MoveL RelTool (p1,78.000000,9.000000,5.500000,\Rx:=0.000000,\Ry:=-0.000000),vel1,zoneval,Extruder\WObj:=Workobject_1;
MoveL RelTool (p1,75.500000,9.000000,5.500000,\Rx:=0.000000,\Ry:=-0.000000),vel1,zoneval,Extruder\WObj:=Workobject_1;
MoveL RelTool (p1,73.000000,9.000000,5.500000,\Rx:=0.000000,\Ry:=-0.000000),vel1,zoneval,Extruder\WObj:=Workobject_1;
MoveL RelTool (p1,70.500000,9.000000,5.500000,\Rx:=0.000000,\Ry:=-0.000000),vel1,zoneval,Extruder\WObj:=Workobject_1;
MoveL RelTool (p1,68.000000,9.000000,5.576212,\Rx:=0.000000,\Ry:=1.027235),vel1,zoneval,Extruder\WObj:=Workobject_1;
MoveL RelTool (p1,65.500000,9.000000,6.601352,\Rx:=0.000000,\Ry:=7.190651),vel1,zoneval,Extruder\WObj:=Workobject_1;
MoveL RelTool (p1,63.000000,9.000000,9.259802,\Rx:=0.000000,\Ry:=10.438096),vel1,zoneval,Extruder\WObj:=Workobject_1;
MoveL RelTool (p1,60.500000,9.000000,11.213438,\Rx:=0.000000,\Ry:=7.277441),vel1,zoneval,Extruder\WObj:=Workobject_1;
MoveL RelTool (p1,58.000000,9.000000,12.567025,\Rx:=0.000000,\Ry:=5.967579),vel1,zoneval,Extruder\WObj:=Workobject_1;
MoveL RelTool (p1,55.500000,9.000000,13.541124,\Rx:=0.000000,\Ry:=4.323199),vel1,zoneval,Extruder\WObj:=Workobject_1;
MoveL RelTool (p1,53.000000,9.000000,14.280270,\Rx:=0.000000,\Ry:=3.233363),vel1,zoneval,Extruder\WObj:=Workobject_1;
MoveL RelTool (p1,50.500000,9.000000,14.829944,\Rx:=0.000000,\Ry:=2.667808),vel1,zoneval,Extruder\WObj:=Workobject_1;
MoveL RelTool (p1,48.000000,9.000000,15.193555,\Rx:=0.000000,\Ry:=1.838961),vel1,zoneval,Extruder\WObj:=Workobject_1;
MoveL RelTool (p1,45.500000,9.000000,15.404325,\Rx:=0.000000,\Ry:=0.957446),vel1,zoneval,Extruder\WObj:=Workobject_1;
MoveL RelTool (p1,43.000000,9.000000,15.486300,\Rx:=0.000000,\Ry:=0.175753),vel1,zoneval,Extruder\WObj:=Workobject_1;
MoveL RelTool (p1,40.500000,9.000000,15.409004,\Rx:=0.000000,\Ry:=-0.609665),vel1,zoneval,Extruder\WObj:=Workobject_1;
MoveL RelTool (p1,38.000000,9.000000,15.198525,\Rx:=0.000000,\Ry:=-1.473255),vel1,zoneval,Extruder\WObj:=Workobject_1;
MoveL RelTool (p1,35.500000,9.000000,14.839102,\Rx:=0.000000,\Ry:=-2.361471),vel1,zoneval,Extruder\WObj:=Workobject_1;
MoveL RelTool (p1,33.000000,9.000000,14.310992,\Rx:=0.000000,\Ry:=-3.310711),vel1,zoneval,Extruder\WObj:=Workobject_1;
MoveL RelTool (p1,30.500000,9.000000,13.585370,\Rx:=0.000000,\Ry:=-4.304408),vel1,zoneval,Extruder\WObj:=Workobject_1;
MoveL RelTool (p1,28.000000,9.000000,12.618075,\Rx:=0.000000,\Ry:=-5.366573),vel1,zoneval,Extruder\WObj:=Workobject_1;
MoveL RelTool (p1,25.500000,9.000000,11.328519,\Rx:=0.000000,\Ry:=-6.568275),vel1,zoneval,Extruder\WObj:=Workobject_1;
MoveL RelTool (p1,23.000000,9.000000,9.422774,\Rx:=0.000000,\Ry:=-9.481583),vel1,zoneval,Extruder\WObj:=Workobject_1;
MoveL RelTool (p1,20.500000,9.000000,6.707804,\Rx:=0.000000,\Ry:=-9.245066),vel1,zoneval,Extruder\WObj:=Workobject_1;
MoveL RelTool (p1,18.000000,9.000000,5.614048,\Rx:=0.000000,\Ry:=-3.081691),vel1,zoneval,Extruder\WObj:=Workobject_1;
MoveL RelTool (p1,15.500000,9.000000,5.500000,\Rx:=0.000000,\Ry:=-0.000000),vel1,zoneval,Extruder\WObj:=Workobject_1;
MoveL RelTool (p1,13.000000,9.000000,5.500000,\Rx:=0.000000,\Ry:=-0.000000),vel1,zoneval,Extruder\WObj:=Workobject_1;
MoveL RelTool (p1,10.500000,9.000000,5.500000,\Rx:=0.000000,\Ry:=-0.000000),vel1,zoneval,Extruder\WObj:=Workobject_1;
MoveL RelTool (p1,8.000000,9.000000,5.500000,\Rx:=0.000000,\Ry:=-0.000000),vel1,zoneval,Extruder\WObj:=Workobject_1;
MoveL RelTool (p1,5.500000,9.000000,5.500000,\Rx:=0.000000,\Ry:=-0.000000),vel1,zoneval,Extruder\WObj:=Workobject_1;
MoveL RelTool (p1,3.000000,9.000000,5.500000,\Rx:=0.000000,\Ry:=-0.000000),vel1,zoneval,Extruder\WObj:=Workobject_1;
MoveL RelTool (p1,5.000000,8.500000,5.500000,\Rx:=0.000000,\Ry:=0.000000),vel1,zoneval,Extruder\WObj:=Workobject_1;
MoveL RelTool (p1,7.500000,8.500000,5.500000,\Rx:=0.000000,\Ry:=0.000000),vel1,zoneval,Extruder\WObj:=Workobject_1;
MoveL RelTool (p1,10.000000,8.500000,5.500000,\Rx:=0.000000,\Ry:=0.000000),vel1,zoneval,Extruder\WObj:=Workobject_1;
MoveL RelTool (p1,12.500000,8.500000,5.500000,\Rx:=0.000000,\Ry:=0.000000),vel1,zoneval,Extruder\WObj:=Workobject_1;
MoveL RelTool (p1,15.000000,8.500000,5.500000,\Rx:=0.000000,\Ry:=0.000000),vel1,zoneval,Extruder\WObj:=Workobject_1;
MoveL RelTool (p1,17.500000,8.500000,5.549338,\Rx:=0.000000,\Ry:=-1.027233),vel1,zoneval,Extruder\WObj:=Workobject_1;
MoveL RelTool (p1,20.000000,8.500000,6.390765,\Rx:=0.000000,\Ry:=-6.482955),vel1,zoneval,Extruder\WObj:=Workobject_1;
MoveL RelTool (p1,22.500000,8.500000,8.916208,\Rx:=0.000000,\Ry:=-11.282192),vel1,zoneval,Extruder\WObj:=Workobject_1;
MoveL RelTool (p1,25.000000,8.500000,11.015814,\Rx:=0.000000,\Ry:=-7.926142),vel1,zoneval,Extruder\WObj:=Workobject_1;
MoveL RelTool (p1,27.500000,8.500000,12.393895,\Rx:=0.000000,\Ry:=-5.366573),vel1,zoneval,Extruder\WObj:=Workobject_1;
MoveL RelTool (p1,30.000000,8.500000,13.409588,\Rx:=0.000000,\Ry:=-4.304408),vel1,zoneval,Extruder\WObj:=Workobject_1;
MoveL RelTool (p1,32.500000,8.500000,14.177969,\Rx:=0.000000,\Ry:=-3.310711),vel1,zoneval,Extruder\WObj:=Workobject_1;
MoveL RelTool (p1,35.000000,8.500000,14.745289,\Rx:=0.000000,\Ry:=-2.361471),vel1,zoneval,Extruder\WObj:=Workobject_1;
MoveL RelTool (p1,37.500000,8.500000,15.140411,\Rx:=0.000000,\Ry:=-1.473255),vel1,zoneval,Extruder\WObj:=Workobject_1;
MoveL RelTool (p1,40.000000,8.500000,15.385044,\Rx:=0.000000,\Ry:=-0.609665),vel1,zoneval,Extruder\WObj:=Workobject_1;
MoveL RelTool (p1,42.500000,8.500000,15.493202,\Rx:=0.000000,\Ry:=-0.313643),vel1,zoneval,Extruder\WObj:=Workobject_1;
MoveL RelTool (p1,45.000000,8.500000,15.441995,\Rx:=0.000000,\Ry:=0.600478),vel1,zoneval,Extruder\WObj:=Workobject_1;
MoveL RelTool (p1,47.500000,8.500000,15.253646,\Rx:=0.000000,\Ry:=0.957446),vel1,zoneval,Extruder\WObj:=Workobject_1;
MoveL RelTool (p1,50.000000,8.500000,14.902666,\Rx:=0.000000,\Ry:=1.838961),vel1,zoneval,Extruder\WObj:=Workobject_1;
MoveL RelTool (p1,52.500000,8.500000,14.391107,\Rx:=0.000000,\Ry:=2.777529),vel1,zoneval,Extruder\WObj:=Workobject_1;
MoveL RelTool (p1,55.000000,8.500000,13.693467,\Rx:=0.000000,\Ry:=3.765598),vel1,zoneval,Extruder\WObj:=Workobject_1;
MoveL RelTool (p1,57.500000,8.500000,12.769306,\Rx:=0.000000,\Ry:=4.809648),vel1,zoneval,Extruder\WObj:=Workobject_1;
MoveL RelTool (p1,60.000000,8.500000,11.535030,\Rx:=0.000000,\Ry:=6.353659),vel1,zoneval,Extruder\WObj:=Workobject_1;
MoveL RelTool (p1,62.500000,8.500000,9.740509,\Rx:=0.000000,\Ry:=8.756273),vel1,zoneval,Extruder\WObj:=Workobject_1;
MoveL RelTool (p1,65.000000,8.500000,7.002928,\Rx:=0.000000,\Ry:=9.759467),vel1,zoneval,Extruder\WObj:=Workobject_1;
MoveL RelTool (p1,67.500000,8.500000,5.696103,\Rx:=0.000000,\Ry:=3.252694),vel1,zoneval,Extruder\WObj:=Workobject_1;
MoveL RelTool (p1,70.000000,8.500000,5.500000,\Rx:=0.000000,\Ry:=0.000000),vel1,zoneval,Extruder\WObj:=Workobject_1;
MoveL RelTool (p1,72.500000,8.500000,5.500000,\Rx:=0.000000,\Ry:=0.000000),vel1,zoneval,Extruder\WObj:=Workobject_1;
MoveL RelTool (p1,75.000000,8.500000,5.500000,\Rx:=0.000000,\Ry:=0.000000),vel1,zoneval,Extruder\WObj:=Workobject_1;
MoveL RelTool (p1,77.500000,8.500000,5.500000,\Rx:=0.000000,\Ry:=0.000000),vel1,zoneval,Extruder\WObj:=Workobject_1;
MoveL RelTool (p1,80.000000,8.500000,5.500000,\Rx:=0.000000,\Ry:=0.000000),vel1,zoneval,Extruder\WObj:=Workobject_1;
MoveL RelTool (p1,82.500000,8.500000,5.500000,\Rx:=0.000000,\Ry:=0.000000),vel1,zoneval,Extruder\WObj:=Workobject_1;
MoveL RelTool (p1,80.500000,8.000000,5.500000,\Rx:=0.000000,\Ry:=-0.000000),vel1,zoneval,Extruder\WObj:=Workobject_1;
MoveL RelTool (p1,78.000000,8.000000,5.500000,\Rx:=0.000000,\Ry:=-0.000000),vel1,zoneval,Extruder\WObj:=Workobject_1;
MoveL RelTool (p1,75.500000,8.000000,5.500000,\Rx:=0.000000,\Ry:=-0.000000),vel1,zoneval,Extruder\WObj:=Workobject_1;
MoveL RelTool (p1,73.000000,8.000000,5.500000,\Rx:=0.000000,\Ry:=-0.000000),vel1,zoneval,Extruder\WObj:=Workobject_1;
MoveL RelTool (p1,70.500000,8.000000,5.500000,\Rx:=0.000000,\Ry:=-0.000000),vel1,zoneval,Extruder\WObj:=Workobject_1;
MoveL RelTool (p1,68.000000,8.000000,5.576212,\Rx:=0.000000,\Ry:=1.027235),vel1,zoneval,Extruder\WObj:=Workobject_1;
MoveL RelTool (p1,65.500000,8.000000,6.601352,\Rx:=0.000000,\Ry:=7.190651),vel1,zoneval,Extruder\WObj:=Workobject_1;
MoveL RelTool (p1,63.000000,8.000000,9.259802,\Rx:=0.000000,\Ry:=10.438096),vel1,zoneval,Extruder\WObj:=Workobject_1;
MoveL RelTool (p1,60.500000,8.000000,11.213438,\Rx:=0.000000,\Ry:=7.277441),vel1,zoneval,Extruder\WObj:=Workobject_1;
MoveL RelTool (p1,58.000000,8.000000,12.567025,\Rx:=0.000000,\Ry:=5.967579),vel1,zoneval,Extruder\WObj:=Workobject_1;
MoveL RelTool (p1,55.500000,8.000000,13.541124,\Rx:=0.000000,\Ry:=4.323199),vel1,zoneval,Extruder\WObj:=Workobject_1;
MoveL RelTool (p1,53.000000,8.000000,14.280270,\Rx:=0.000000,\Ry:=3.233363),vel1,zoneval,Extruder\WObj:=Workobject_1;
MoveL RelTool (p1,50.500000,8.000000,14.829944,\Rx:=0.000000,\Ry:=2.667808),vel1,zoneval,Extruder\WObj:=Workobject_1;
MoveL RelTool (p1,48.000000,8.000000,15.193555,\Rx:=0.000000,\Ry:=1.838961),vel1,zoneval,Extruder\WObj:=Workobject_1;
MoveL RelTool (p1,45.500000,8.000000,15.404325,\Rx:=0.000000,\Ry:=0.957446),vel1,zoneval,Extruder\WObj:=Workobject_1;
MoveL RelTool (p1,43.000000,8.000000,15.486300,\Rx:=0.000000,\Ry:=0.175753),vel1,zoneval,Extruder\WObj:=Workobject_1;
MoveL RelTool (p1,40.500000,8.000000,15.409004,\Rx:=0.000000,\Ry:=-0.609665),vel1,zoneval,Extruder\WObj:=Workobject_1;
MoveL RelTool (p1,38.000000,8.000000,15.198525,\Rx:=0.000000,\Ry:=-1.473255),vel1,zoneval,Extruder\WObj:=Workobject_1;
MoveL RelTool (p1,35.500000,8.000000,14.839102,\Rx:=0.000000,\Ry:=-2.361471),vel1,zoneval,Extruder\WObj:=Workobject_1;
MoveL RelTool (p1,33.000000,8.000000,14.310992,\Rx:=0.000000,\Ry:=-3.310711),vel1,zoneval,Extruder\WObj:=Workobject_1;
MoveL RelTool (p1,30.500000,8.000000,13.585370,\Rx:=0.000000,\Ry:=-4.304408),vel1,zoneval,Extruder\WObj:=Workobject_1;
MoveL RelTool (p1,28.000000,8.000000,12.618075,\Rx:=0.000000,\Ry:=-5.366573),vel1,zoneval,Extruder\WObj:=Workobject_1;
MoveL RelTool (p1,25.500000,8.000000,11.328519,\Rx:=0.000000,\Ry:=-6.568275),vel1,zoneval,Extruder\WObj:=Workobject_1;
MoveL RelTool (p1,23.000000,8.000000,9.422774,\Rx:=0.000000,\Ry:=-9.481583),vel1,zoneval,Extruder\WObj:=Workobject_1;
MoveL RelTool (p1,20.500000,8.000000,6.707804,\Rx:=0.000000,\Ry:=-9.245066),vel1,zoneval,Extruder\WObj:=Workobject_1;
MoveL RelTool (p1,18.000000,8.000000,5.614048,\Rx:=0.000000,\Ry:=-3.081691),vel1,zoneval,Extruder\WObj:=Workobject_1;
MoveL RelTool (p1,15.500000,8.000000,5.500000,\Rx:=0.000000,\Ry:=-0.000000),vel1,zoneval,Extruder\WObj:=Workobject_1;
MoveL RelTool (p1,13.000000,8.000000,5.500000,\Rx:=0.000000,\Ry:=-0.000000),vel1,zoneval,Extruder\WObj:=Workobject_1;
MoveL RelTool (p1,10.500000,8.000000,5.500000,\Rx:=0.000000,\Ry:=-0.000000),vel1,zoneval,Extruder\WObj:=Workobject_1;
MoveL RelTool (p1,8.000000,8.000000,5.500000,\Rx:=0.000000,\Ry:=-0.000000),vel1,zoneval,Extruder\WObj:=Workobject_1;
MoveL RelTool (p1,5.500000,8.000000,5.500000,\Rx:=0.000000,\Ry:=-0.000000),vel1,zoneval,Extruder\WObj:=Workobject_1;
MoveL RelTool (p1,3.000000,8.000000,5.500000,\Rx:=0.000000,\Ry:=-0.000000),vel1,zoneval,Extruder\WObj:=Workobject_1;
MoveL RelTool (p1,5.000000,7.500000,5.500000,\Rx:=0.000000,\Ry:=0.000000),vel1,zoneval,Extruder\WObj:=Workobject_1;
MoveL RelTool (p1,7.500000,7.500000,5.500000,\Rx:=0.000000,\Ry:=0.000000),vel1,zoneval,Extruder\WObj:=Workobject_1;
MoveL RelTool (p1,10.000000,7.500000,5.500000,\Rx:=0.000000,\Ry:=0.000000),vel1,zoneval,Extruder\WObj:=Workobject_1;
MoveL RelTool (p1,12.500000,7.500000,5.500000,\Rx:=0.000000,\Ry:=0.000000),vel1,zoneval,Extruder\WObj:=Workobject_1;
MoveL RelTool (p1,15.000000,7.500000,5.500000,\Rx:=0.000000,\Ry:=0.000000),vel1,zoneval,Extruder\WObj:=Workobject_1;
MoveL RelTool (p1,17.500000,7.500000,5.549338,\Rx:=0.000000,\Ry:=-1.027233),vel1,zoneval,Extruder\WObj:=Workobject_1;
MoveL RelTool (p1,20.000000,7.500000,6.390765,\Rx:=0.000000,\Ry:=-6.482955),vel1,zoneval,Extruder\WObj:=Workobject_1;
MoveL RelTool (p1,22.500000,7.500000,8.916208,\Rx:=0.000000,\Ry:=-11.282192),vel1,zoneval,Extruder\WObj:=Workobject_1;
MoveL RelTool (p1,25.000000,7.500000,11.015814,\Rx:=0.000000,\Ry:=-7.926142),vel1,zoneval,Extruder\WObj:=Workobject_1;
MoveL RelTool (p1,27.500000,7.500000,12.393895,\Rx:=0.000000,\Ry:=-5.366573),vel1,zoneval,Extruder\WObj:=Workobject_1;
MoveL RelTool (p1,30.000000,7.500000,13.409588,\Rx:=0.000000,\Ry:=-4.304408),vel1,zoneval,Extruder\WObj:=Workobject_1;
MoveL RelTool (p1,32.500000,7.500000,14.177969,\Rx:=0.000000,\Ry:=-3.310711),vel1,zoneval,Extruder\WObj:=Workobject_1;
MoveL RelTool (p1,35.000000,7.500000,14.745289,\Rx:=0.000000,\Ry:=-2.361471),vel1,zoneval,Extruder\WObj:=Workobject_1;
MoveL RelTool (p1,37.500000,7.500000,15.140411,\Rx:=0.000000,\Ry:=-1.473255),vel1,zoneval,Extruder\WObj:=Workobject_1;
MoveL RelTool (p1,40.000000,7.500000,15.385044,\Rx:=0.000000,\Ry:=-0.609665),vel1,zoneval,Extruder\WObj:=Workobject_1;
MoveL RelTool (p1,42.500000,7.500000,15.493202,\Rx:=0.000000,\Ry:=-0.313643),vel1,zoneval,Extruder\WObj:=Workobject_1;
MoveL RelTool (p1,45.000000,7.500000,15.441995,\Rx:=0.000000,\Ry:=0.600478),vel1,zoneval,Extruder\WObj:=Workobject_1;
MoveL RelTool (p1,47.500000,7.500000,15.253646,\Rx:=0.000000,\Ry:=0.957446),vel1,zoneval,Extruder\WObj:=Workobject_1;
MoveL RelTool (p1,50.000000,7.500000,14.902666,\Rx:=0.000000,\Ry:=1.838961),vel1,zoneval,Extruder\WObj:=Workobject_1;
MoveL RelTool (p1,52.500000,7.500000,14.391107,\Rx:=0.000000,\Ry:=2.777529),vel1,zoneval,Extruder\WObj:=Workobject_1;
MoveL RelTool (p1,55.000000,7.500000,13.693467,\Rx:=0.000000,\Ry:=3.765598),vel1,zoneval,Extruder\WObj:=Workobject_1;
MoveL RelTool (p1,57.500000,7.500000,12.769306,\Rx:=0.000000,\Ry:=4.809648),vel1,zoneval,Extruder\WObj:=Workobject_1;
MoveL RelTool (p1,60.000000,7.500000,11.535030,\Rx:=0.000000,\Ry:=6.353659),vel1,zoneval,Extruder\WObj:=Workobject_1;
MoveL RelTool (p1,62.500000,7.500000,9.740509,\Rx:=0.000000,\Ry:=8.756273),vel1,zoneval,Extruder\WObj:=Workobject_1;
MoveL RelTool (p1,65.000000,7.500000,7.002928,\Rx:=0.000000,\Ry:=9.759467),vel1,zoneval,Extruder\WObj:=Workobject_1;
MoveL RelTool (p1,67.500000,7.500000,5.696103,\Rx:=0.000000,\Ry:=3.252694),vel1,zoneval,Extruder\WObj:=Workobject_1;
MoveL RelTool (p1,70.000000,7.500000,5.500000,\Rx:=0.000000,\Ry:=0.000000),vel1,zoneval,Extruder\WObj:=Workobject_1;
MoveL RelTool (p1,72.500000,7.500000,5.500000,\Rx:=0.000000,\Ry:=0.000000),vel1,zoneval,Extruder\WObj:=Workobject_1;
MoveL RelTool (p1,75.000000,7.500000,5.500000,\Rx:=0.000000,\Ry:=0.000000),vel1,zoneval,Extruder\WObj:=Workobject_1;
MoveL RelTool (p1,77.500000,7.500000,5.500000,\Rx:=0.000000,\Ry:=0.000000),vel1,zoneval,Extruder\WObj:=Workobject_1;
MoveL RelTool (p1,80.000000,7.500000,5.500000,\Rx:=0.000000,\Ry:=0.000000),vel1,zoneval,Extruder\WObj:=Workobject_1;
MoveL RelTool (p1,82.500000,7.500000,5.500000,\Rx:=0.000000,\Ry:=0.000000),vel1,zoneval,Extruder\WObj:=Workobject_1;
MoveL RelTool (p1,80.500000,7.000000,5.500000,\Rx:=0.000000,\Ry:=-0.000000),vel1,zoneval,Extruder\WObj:=Workobject_1;
MoveL RelTool (p1,78.000000,7.000000,5.500000,\Rx:=0.000000,\Ry:=-0.000000),vel1,zoneval,Extruder\WObj:=Workobject_1;
MoveL RelTool (p1,75.500000,7.000000,5.500000,\Rx:=0.000000,\Ry:=-0.000000),vel1,zoneval,Extruder\WObj:=Workobject_1;
MoveL RelTool (p1,73.000000,7.000000,5.500000,\Rx:=0.000000,\Ry:=-0.000000),vel1,zoneval,Extruder\WObj:=Workobject_1;
MoveL RelTool (p1,70.500000,7.000000,5.500000,\Rx:=0.000000,\Ry:=-0.000000),vel1,zoneval,Extruder\WObj:=Workobject_1;
MoveL RelTool (p1,68.000000,7.000000,5.576212,\Rx:=0.000000,\Ry:=1.027235),vel1,zoneval,Extruder\WObj:=Workobject_1;
MoveL RelTool (p1,65.500000,7.000000,6.601352,\Rx:=0.000000,\Ry:=7.190651),vel1,zoneval,Extruder\WObj:=Workobject_1;
MoveL RelTool (p1,63.000000,7.000000,9.259802,\Rx:=0.000000,\Ry:=10.438096),vel1,zoneval,Extruder\WObj:=Workobject_1;
MoveL RelTool (p1,60.500000,7.000000,11.213438,\Rx:=0.000000,\Ry:=7.277441),vel1,zoneval,Extruder\WObj:=Workobject_1;
MoveL RelTool (p1,58.000000,7.000000,12.567025,\Rx:=0.000000,\Ry:=5.967579),vel1,zoneval,Extruder\WObj:=Workobject_1;
MoveL RelTool (p1,55.500000,7.000000,13.541124,\Rx:=0.000000,\Ry:=4.323199),vel1,zoneval,Extruder\WObj:=Workobject_1;
MoveL RelTool (p1,53.000000,7.000000,14.280270,\Rx:=0.000000,\Ry:=3.233363),vel1,zoneval,Extruder\WObj:=Workobject_1;
MoveL RelTool (p1,50.500000,7.000000,14.829944,\Rx:=0.000000,\Ry:=2.667808),vel1,zoneval,Extruder\WObj:=Workobject_1;
MoveL RelTool (p1,48.000000,7.000000,15.193555,\Rx:=0.000000,\Ry:=1.838961),vel1,zoneval,Extruder\WObj:=Workobject_1;
MoveL RelTool (p1,45.500000,7.000000,15.404325,\Rx:=0.000000,\Ry:=0.957446),vel1,zoneval,Extruder\WObj:=Workobject_1;
MoveL RelTool (p1,43.000000,7.000000,15.486300,\Rx:=0.000000,\Ry:=0.175753),vel1,zoneval,Extruder\WObj:=Workobject_1;
MoveL RelTool (p1,40.500000,7.000000,15.409004,\Rx:=0.000000,\Ry:=-0.609665),vel1,zoneval,Extruder\WObj:=Workobject_1;
MoveL RelTool (p1,38.000000,7.000000,15.198525,\Rx:=0.000000,\Ry:=-1.473255),vel1,zoneval,Extruder\WObj:=Workobject_1;
MoveL RelTool (p1,35.500000,7.000000,14.839102,\Rx:=0.000000,\Ry:=-2.361471),vel1,zoneval,Extruder\WObj:=Workobject_1;
MoveL RelTool (p1,33.000000,7.000000,14.310992,\Rx:=0.000000,\Ry:=-3.310711),vel1,zoneval,Extruder\WObj:=Workobject_1;
MoveL RelTool (p1,30.500000,7.000000,13.585370,\Rx:=0.000000,\Ry:=-4.304408),vel1,zoneval,Extruder\WObj:=Workobject_1;
MoveL RelTool (p1,28.000000,7.000000,12.618075,\Rx:=0.000000,\Ry:=-5.366573),vel1,zoneval,Extruder\WObj:=Workobject_1;
MoveL RelTool (p1,25.500000,7.000000,11.328519,\Rx:=0.000000,\Ry:=-6.568275),vel1,zoneval,Extruder\WObj:=Workobject_1;
MoveL RelTool (p1,23.000000,7.000000,9.422774,\Rx:=0.000000,\Ry:=-9.481583),vel1,zoneval,Extruder\WObj:=Workobject_1;
MoveL RelTool (p1,20.500000,7.000000,6.707804,\Rx:=0.000000,\Ry:=-9.245066),vel1,zoneval,Extruder\WObj:=Workobject_1;
MoveL RelTool (p1,18.000000,7.000000,5.614048,\Rx:=0.000000,\Ry:=-3.081691),vel1,zoneval,Extruder\WObj:=Workobject_1;
MoveL RelTool (p1,15.500000,7.000000,5.500000,\Rx:=0.000000,\Ry:=-0.000000),vel1,zoneval,Extruder\WObj:=Workobject_1;
MoveL RelTool (p1,13.000000,7.000000,5.500000,\Rx:=0.000000,\Ry:=-0.000000),vel1,zoneval,Extruder\WObj:=Workobject_1;
MoveL RelTool (p1,10.500000,7.000000,5.500000,\Rx:=0.000000,\Ry:=-0.000000),vel1,zoneval,Extruder\WObj:=Workobject_1;
MoveL RelTool (p1,8.000000,7.000000,5.500000,\Rx:=0.000000,\Ry:=-0.000000),vel1,zoneval,Extruder\WObj:=Workobject_1;
MoveL RelTool (p1,5.500000,7.000000,5.500000,\Rx:=0.000000,\Ry:=-0.000000),vel1,zoneval,Extruder\WObj:=Workobject_1;
MoveL RelTool (p1,3.000000,7.000000,5.500000,\Rx:=0.000000,\Ry:=-0.000000),vel1,zoneval,Extruder\WObj:=Workobject_1;
MoveL RelTool (p1,5.000000,6.500000,5.500000,\Rx:=0.000000,\Ry:=0.000000),vel1,zoneval,Extruder\WObj:=Workobject_1;
MoveL RelTool (p1,7.500000,6.500000,5.500000,\Rx:=0.000000,\Ry:=0.000000),vel1,zoneval,Extruder\WObj:=Workobject_1;
MoveL RelTool (p1,10.000000,6.500000,5.500000,\Rx:=0.000000,\Ry:=0.000000),vel1,zoneval,Extruder\WObj:=Workobject_1;
MoveL RelTool (p1,12.500000,6.500000,5.500000,\Rx:=0.000000,\Ry:=0.000000),vel1,zoneval,Extruder\WObj:=Workobject_1;
MoveL RelTool (p1,15.000000,6.500000,5.500000,\Rx:=0.000000,\Ry:=0.000000),vel1,zoneval,Extruder\WObj:=Workobject_1;
MoveL RelTool (p1,17.500000,6.500000,5.549338,\Rx:=0.000000,\Ry:=-1.027233),vel1,zoneval,Extruder\WObj:=Workobject_1;
MoveL RelTool (p1,20.000000,6.500000,6.390765,\Rx:=0.000000,\Ry:=-6.482955),vel1,zoneval,Extruder\WObj:=Workobject_1;
MoveL RelTool (p1,22.500000,6.500000,8.916208,\Rx:=0.000000,\Ry:=-11.282192),vel1,zoneval,Extruder\WObj:=Workobject_1;
MoveL RelTool (p1,25.000000,6.500000,11.015814,\Rx:=0.000000,\Ry:=-7.926142),vel1,zoneval,Extruder\WObj:=Workobject_1;
MoveL RelTool (p1,27.500000,6.500000,12.393895,\Rx:=0.000000,\Ry:=-5.366573),vel1,zoneval,Extruder\WObj:=Workobject_1;
MoveL RelTool (p1,30.000000,6.500000,13.409588,\Rx:=0.000000,\Ry:=-4.304408),vel1,zoneval,Extruder\WObj:=Workobject_1;
MoveL RelTool (p1,32.500000,6.500000,14.177969,\Rx:=0.000000,\Ry:=-3.310711),vel1,zoneval,Extruder\WObj:=Workobject_1;
MoveL RelTool (p1,35.000000,6.500000,14.745289,\Rx:=0.000000,\Ry:=-2.361471),vel1,zoneval,Extruder\WObj:=Workobject_1;
MoveL RelTool (p1,37.500000,6.500000,15.140411,\Rx:=0.000000,\Ry:=-1.473255),vel1,zoneval,Extruder\WObj:=Workobject_1;
MoveL RelTool (p1,40.000000,6.500000,15.385044,\Rx:=0.000000,\Ry:=-0.609665),vel1,zoneval,Extruder\WObj:=Workobject_1;
MoveL RelTool (p1,42.500000,6.500000,15.493202,\Rx:=0.000000,\Ry:=-0.313643),vel1,zoneval,Extruder\WObj:=Workobject_1;
MoveL RelTool (p1,45.000000,6.500000,15.441995,\Rx:=0.000000,\Ry:=0.600478),vel1,zoneval,Extruder\WObj:=Workobject_1;
MoveL RelTool (p1,47.500000,6.500000,15.253646,\Rx:=0.000000,\Ry:=0.957446),vel1,zoneval,Extruder\WObj:=Workobject_1;
MoveL RelTool (p1,50.000000,6.500000,14.902666,\Rx:=0.000000,\Ry:=1.838961),vel1,zoneval,Extruder\WObj:=Workobject_1;
MoveL RelTool (p1,52.500000,6.500000,14.391107,\Rx:=0.000000,\Ry:=2.777529),vel1,zoneval,Extruder\WObj:=Workobject_1;
MoveL RelTool (p1,55.000000,6.500000,13.693467,\Rx:=0.000000,\Ry:=3.765598),vel1,zoneval,Extruder\WObj:=Workobject_1;
MoveL RelTool (p1,57.500000,6.500000,12.769306,\Rx:=0.000000,\Ry:=4.809648),vel1,zoneval,Extruder\WObj:=Workobject_1;
MoveL RelTool (p1,60.000000,6.500000,11.535030,\Rx:=0.000000,\Ry:=6.353659),vel1,zoneval,Extruder\WObj:=Workobject_1;
MoveL RelTool (p1,62.500000,6.500000,9.740509,\Rx:=0.000000,\Ry:=8.756273),vel1,zoneval,Extruder\WObj:=Workobject_1;
MoveL RelTool (p1,65.000000,6.500000,7.002928,\Rx:=0.000000,\Ry:=9.759467),vel1,zoneval,Extruder\WObj:=Workobject_1;
MoveL RelTool (p1,67.500000,6.500000,5.696103,\Rx:=0.000000,\Ry:=3.252694),vel1,zoneval,Extruder\WObj:=Workobject_1;
MoveL RelTool (p1,70.000000,6.500000,5.500000,\Rx:=0.000000,\Ry:=0.000000),vel1,zoneval,Extruder\WObj:=Workobject_1;
MoveL RelTool (p1,72.500000,6.500000,5.500000,\Rx:=0.000000,\Ry:=0.000000),vel1,zoneval,Extruder\WObj:=Workobject_1;
MoveL RelTool (p1,75.000000,6.500000,5.500000,\Rx:=0.000000,\Ry:=0.000000),vel1,zoneval,Extruder\WObj:=Workobject_1;
MoveL RelTool (p1,77.500000,6.500000,5.500000,\Rx:=0.000000,\Ry:=0.000000),vel1,zoneval,Extruder\WObj:=Workobject_1;
MoveL RelTool (p1,80.000000,6.500000,5.500000,\Rx:=0.000000,\Ry:=0.000000),vel1,zoneval,Extruder\WObj:=Workobject_1;
MoveL RelTool (p1,82.500000,6.500000,5.500000,\Rx:=0.000000,\Ry:=0.000000),vel1,zoneval,Extruder\WObj:=Workobject_1;
MoveL RelTool (p1,80.500000,6.000000,5.500000,\Rx:=0.000000,\Ry:=-0.000000),vel1,zoneval,Extruder\WObj:=Workobject_1;
MoveL RelTool (p1,78.000000,6.000000,5.500000,\Rx:=0.000000,\Ry:=-0.000000),vel1,zoneval,Extruder\WObj:=Workobject_1;
MoveL RelTool (p1,75.500000,6.000000,5.500000,\Rx:=0.000000,\Ry:=-0.000000),vel1,zoneval,Extruder\WObj:=Workobject_1;
MoveL RelTool (p1,73.000000,6.000000,5.500000,\Rx:=0.000000,\Ry:=-0.000000),vel1,zoneval,Extruder\WObj:=Workobject_1;
MoveL RelTool (p1,70.500000,6.000000,5.500000,\Rx:=0.000000,\Ry:=-0.000000),vel1,zoneval,Extruder\WObj:=Workobject_1;
MoveL RelTool (p1,68.000000,6.000000,5.576212,\Rx:=0.000000,\Ry:=1.027235),vel1,zoneval,Extruder\WObj:=Workobject_1;
MoveL RelTool (p1,65.500000,6.000000,6.601352,\Rx:=0.000000,\Ry:=7.190651),vel1,zoneval,Extruder\WObj:=Workobject_1;
MoveL RelTool (p1,63.000000,6.000000,9.259802,\Rx:=0.000000,\Ry:=10.438096),vel1,zoneval,Extruder\WObj:=Workobject_1;
MoveL RelTool (p1,60.500000,6.000000,11.213438,\Rx:=0.000000,\Ry:=7.277441),vel1,zoneval,Extruder\WObj:=Workobject_1;
MoveL RelTool (p1,58.000000,6.000000,12.567025,\Rx:=0.000000,\Ry:=5.967579),vel1,zoneval,Extruder\WObj:=Workobject_1;
MoveL RelTool (p1,55.500000,6.000000,13.541124,\Rx:=0.000000,\Ry:=4.323199),vel1,zoneval,Extruder\WObj:=Workobject_1;
MoveL RelTool (p1,53.000000,6.000000,14.280270,\Rx:=0.000000,\Ry:=3.233363),vel1,zoneval,Extruder\WObj:=Workobject_1;
MoveL RelTool (p1,50.500000,6.000000,14.829944,\Rx:=0.000000,\Ry:=2.667808),vel1,zoneval,Extruder\WObj:=Workobject_1;
MoveL RelTool (p1,48.000000,6.000000,15.193555,\Rx:=0.000000,\Ry:=1.838961),vel1,zoneval,Extruder\WObj:=Workobject_1;
MoveL RelTool (p1,45.500000,6.000000,15.404325,\Rx:=0.000000,\Ry:=0.957446),vel1,zoneval,Extruder\WObj:=Workobject_1;
MoveL RelTool (p1,43.000000,6.000000,15.486300,\Rx:=0.000000,\Ry:=0.175753),vel1,zoneval,Extruder\WObj:=Workobject_1;
MoveL RelTool (p1,40.500000,6.000000,15.409004,\Rx:=0.000000,\Ry:=-0.609665),vel1,zoneval,Extruder\WObj:=Workobject_1;
MoveL RelTool (p1,38.000000,6.000000,15.198525,\Rx:=0.000000,\Ry:=-1.473255),vel1,zoneval,Extruder\WObj:=Workobject_1;
MoveL RelTool (p1,35.500000,6.000000,14.839102,\Rx:=0.000000,\Ry:=-2.361471),vel1,zoneval,Extruder\WObj:=Workobject_1;
MoveL RelTool (p1,33.000000,6.000000,14.310992,\Rx:=0.000000,\Ry:=-3.310711),vel1,zoneval,Extruder\WObj:=Workobject_1;
MoveL RelTool (p1,30.500000,6.000000,13.585370,\Rx:=0.000000,\Ry:=-4.304408),vel1,zoneval,Extruder\WObj:=Workobject_1;
MoveL RelTool (p1,28.000000,6.000000,12.618075,\Rx:=0.000000,\Ry:=-5.366573),vel1,zoneval,Extruder\WObj:=Workobject_1;
MoveL RelTool (p1,25.500000,6.000000,11.328519,\Rx:=0.000000,\Ry:=-6.568275),vel1,zoneval,Extruder\WObj:=Workobject_1;
MoveL RelTool (p1,23.000000,6.000000,9.422774,\Rx:=0.000000,\Ry:=-9.481583),vel1,zoneval,Extruder\WObj:=Workobject_1;
MoveL RelTool (p1,20.500000,6.000000,6.707804,\Rx:=0.000000,\Ry:=-9.245066),vel1,zoneval,Extruder\WObj:=Workobject_1;
MoveL RelTool (p1,18.000000,6.000000,5.614048,\Rx:=0.000000,\Ry:=-3.081691),vel1,zoneval,Extruder\WObj:=Workobject_1;
MoveL RelTool (p1,15.500000,6.000000,5.500000,\Rx:=0.000000,\Ry:=-0.000000),vel1,zoneval,Extruder\WObj:=Workobject_1;
MoveL RelTool (p1,13.000000,6.000000,5.500000,\Rx:=0.000000,\Ry:=-0.000000),vel1,zoneval,Extruder\WObj:=Workobject_1;
MoveL RelTool (p1,10.500000,6.000000,5.500000,\Rx:=0.000000,\Ry:=-0.000000),vel1,zoneval,Extruder\WObj:=Workobject_1;
MoveL RelTool (p1,8.000000,6.000000,5.500000,\Rx:=0.000000,\Ry:=-0.000000),vel1,zoneval,Extruder\WObj:=Workobject_1;
MoveL RelTool (p1,5.500000,6.000000,5.500000,\Rx:=0.000000,\Ry:=-0.000000),vel1,zoneval,Extruder\WObj:=Workobject_1;
MoveL RelTool (p1,3.000000,6.000000,5.500000,\Rx:=0.000000,\Ry:=-0.000000),vel1,zoneval,Extruder\WObj:=Workobject_1;
MoveL RelTool (p1,5.000000,5.500000,5.500000,\Rx:=0.000000,\Ry:=0.000000),vel1,zoneval,Extruder\WObj:=Workobject_1;
MoveL RelTool (p1,7.500000,5.500000,5.500000,\Rx:=0.000000,\Ry:=0.000000),vel1,zoneval,Extruder\WObj:=Workobject_1;
MoveL RelTool (p1,10.000000,5.500000,5.500000,\Rx:=0.000000,\Ry:=0.000000),vel1,zoneval,Extruder\WObj:=Workobject_1;
MoveL RelTool (p1,12.500000,5.500000,5.500000,\Rx:=0.000000,\Ry:=0.000000),vel1,zoneval,Extruder\WObj:=Workobject_1;
MoveL RelTool (p1,15.000000,5.500000,5.500000,\Rx:=0.000000,\Ry:=0.000000),vel1,zoneval,Extruder\WObj:=Workobject_1;
MoveL RelTool (p1,17.500000,5.500000,5.549338,\Rx:=0.000000,\Ry:=-1.027233),vel1,zoneval,Extruder\WObj:=Workobject_1;
MoveL RelTool (p1,20.000000,5.500000,6.390765,\Rx:=0.000000,\Ry:=-6.482955),vel1,zoneval,Extruder\WObj:=Workobject_1;
MoveL RelTool (p1,22.500000,5.500000,8.916208,\Rx:=0.000000,\Ry:=-11.282192),vel1,zoneval,Extruder\WObj:=Workobject_1;
MoveL RelTool (p1,25.000000,5.500000,11.015814,\Rx:=0.000000,\Ry:=-7.926142),vel1,zoneval,Extruder\WObj:=Workobject_1;
MoveL RelTool (p1,27.500000,5.500000,12.393895,\Rx:=0.000000,\Ry:=-5.366573),vel1,zoneval,Extruder\WObj:=Workobject_1;
MoveL RelTool (p1,30.000000,5.500000,13.409588,\Rx:=0.000000,\Ry:=-4.304408),vel1,zoneval,Extruder\WObj:=Workobject_1;
MoveL RelTool (p1,32.500000,5.500000,14.177969,\Rx:=0.000000,\Ry:=-3.310711),vel1,zoneval,Extruder\WObj:=Workobject_1;
MoveL RelTool (p1,35.000000,5.500000,14.745289,\Rx:=0.000000,\Ry:=-2.361471),vel1,zoneval,Extruder\WObj:=Workobject_1;
MoveL RelTool (p1,37.500000,5.500000,15.140411,\Rx:=0.000000,\Ry:=-1.473255),vel1,zoneval,Extruder\WObj:=Workobject_1;
MoveL RelTool (p1,40.000000,5.500000,15.385044,\Rx:=0.000000,\Ry:=-0.609665),vel1,zoneval,Extruder\WObj:=Workobject_1;
MoveL RelTool (p1,42.500000,5.500000,15.493202,\Rx:=0.000000,\Ry:=-0.313643),vel1,zoneval,Extruder\WObj:=Workobject_1;
MoveL RelTool (p1,45.000000,5.500000,15.441995,\Rx:=0.000000,\Ry:=0.600478),vel1,zoneval,Extruder\WObj:=Workobject_1;
MoveL RelTool (p1,47.500000,5.500000,15.253646,\Rx:=0.000000,\Ry:=0.957446),vel1,zoneval,Extruder\WObj:=Workobject_1;
MoveL RelTool (p1,50.000000,5.500000,14.902666,\Rx:=0.000000,\Ry:=1.838961),vel1,zoneval,Extruder\WObj:=Workobject_1;
MoveL RelTool (p1,52.500000,5.500000,14.391107,\Rx:=0.000000,\Ry:=2.777529),vel1,zoneval,Extruder\WObj:=Workobject_1;
MoveL RelTool (p1,55.000000,5.500000,13.693467,\Rx:=0.000000,\Ry:=3.765598),vel1,zoneval,Extruder\WObj:=Workobject_1;
MoveL RelTool (p1,57.500000,5.500000,12.769306,\Rx:=0.000000,\Ry:=4.809648),vel1,zoneval,Extruder\WObj:=Workobject_1;
MoveL RelTool (p1,60.000000,5.500000,11.535030,\Rx:=0.000000,\Ry:=6.353659),vel1,zoneval,Extruder\WObj:=Workobject_1;
MoveL RelTool (p1,62.500000,5.500000,9.740509,\Rx:=0.000000,\Ry:=8.756273),vel1,zoneval,Extruder\WObj:=Workobject_1;
MoveL RelTool (p1,65.000000,5.500000,7.002928,\Rx:=0.000000,\Ry:=9.759467),vel1,zoneval,Extruder\WObj:=Workobject_1;
MoveL RelTool (p1,67.500000,5.500000,5.696103,\Rx:=0.000000,\Ry:=3.252694),vel1,zoneval,Extruder\WObj:=Workobject_1;
MoveL RelTool (p1,70.000000,5.500000,5.500000,\Rx:=0.000000,\Ry:=0.000000),vel1,zoneval,Extruder\WObj:=Workobject_1;
MoveL RelTool (p1,72.500000,5.500000,5.500000,\Rx:=0.000000,\Ry:=0.000000),vel1,zoneval,Extruder\WObj:=Workobject_1;
MoveL RelTool (p1,75.000000,5.500000,5.500000,\Rx:=0.000000,\Ry:=0.000000),vel1,zoneval,Extruder\WObj:=Workobject_1;
MoveL RelTool (p1,77.500000,5.500000,5.500000,\Rx:=0.000000,\Ry:=0.000000),vel1,zoneval,Extruder\WObj:=Workobject_1;
MoveL RelTool (p1,80.000000,5.500000,5.500000,\Rx:=0.000000,\Ry:=0.000000),vel1,zoneval,Extruder\WObj:=Workobject_1;
MoveL RelTool (p1,82.500000,5.500000,5.500000,\Rx:=0.000000,\Ry:=0.000000),vel1,zoneval,Extruder\WObj:=Workobject_1;
MoveL RelTool (p1,80.500000,5.000000,5.500000,\Rx:=0.000000,\Ry:=-0.000000),vel1,zoneval,Extruder\WObj:=Workobject_1;
MoveL RelTool (p1,78.000000,5.000000,5.500000,\Rx:=0.000000,\Ry:=-0.000000),vel1,zoneval,Extruder\WObj:=Workobject_1;
MoveL RelTool (p1,75.500000,5.000000,5.500000,\Rx:=0.000000,\Ry:=-0.000000),vel1,zoneval,Extruder\WObj:=Workobject_1;
MoveL RelTool (p1,73.000000,5.000000,5.500000,\Rx:=0.000000,\Ry:=-0.000000),vel1,zoneval,Extruder\WObj:=Workobject_1;
MoveL RelTool (p1,70.500000,5.000000,5.500000,\Rx:=0.000000,\Ry:=-0.000000),vel1,zoneval,Extruder\WObj:=Workobject_1;
MoveL RelTool (p1,68.000000,5.000000,5.576212,\Rx:=0.000000,\Ry:=1.027235),vel1,zoneval,Extruder\WObj:=Workobject_1;
MoveL RelTool (p1,65.500000,5.000000,6.601352,\Rx:=0.000000,\Ry:=7.190651),vel1,zoneval,Extruder\WObj:=Workobject_1;
MoveL RelTool (p1,63.000000,5.000000,9.259802,\Rx:=0.000000,\Ry:=10.438096),vel1,zoneval,Extruder\WObj:=Workobject_1;
MoveL RelTool (p1,60.500000,5.000000,11.213438,\Rx:=0.000000,\Ry:=7.277441),vel1,zoneval,Extruder\WObj:=Workobject_1;
MoveL RelTool (p1,58.000000,5.000000,12.567025,\Rx:=0.000000,\Ry:=5.967579),vel1,zoneval,Extruder\WObj:=Workobject_1;
MoveL RelTool (p1,55.500000,5.000000,13.541124,\Rx:=0.000000,\Ry:=4.323199),vel1,zoneval,Extruder\WObj:=Workobject_1;
MoveL RelTool (p1,53.000000,5.000000,14.280270,\Rx:=0.000000,\Ry:=3.233363),vel1,zoneval,Extruder\WObj:=Workobject_1;
MoveL RelTool (p1,50.500000,5.000000,14.829944,\Rx:=0.000000,\Ry:=2.667808),vel1,zoneval,Extruder\WObj:=Workobject_1;
MoveL RelTool (p1,48.000000,5.000000,15.193555,\Rx:=0.000000,\Ry:=1.838961),vel1,zoneval,Extruder\WObj:=Workobject_1;
MoveL RelTool (p1,45.500000,5.000000,15.404325,\Rx:=0.000000,\Ry:=0.957446),vel1,zoneval,Extruder\WObj:=Workobject_1;
MoveL RelTool (p1,43.000000,5.000000,15.486300,\Rx:=0.000000,\Ry:=0.175753),vel1,zoneval,Extruder\WObj:=Workobject_1;
MoveL RelTool (p1,40.500000,5.000000,15.409004,\Rx:=0.000000,\Ry:=-0.609665),vel1,zoneval,Extruder\WObj:=Workobject_1;
MoveL RelTool (p1,38.000000,5.000000,15.198525,\Rx:=0.000000,\Ry:=-1.473255),vel1,zoneval,Extruder\WObj:=Workobject_1;
MoveL RelTool (p1,35.500000,5.000000,14.839102,\Rx:=0.000000,\Ry:=-2.361471),vel1,zoneval,Extruder\WObj:=Workobject_1;
MoveL RelTool (p1,33.000000,5.000000,14.310992,\Rx:=0.000000,\Ry:=-3.310711),vel1,zoneval,Extruder\WObj:=Workobject_1;
MoveL RelTool (p1,30.500000,5.000000,13.585370,\Rx:=0.000000,\Ry:=-4.304408),vel1,zoneval,Extruder\WObj:=Workobject_1;
MoveL RelTool (p1,28.000000,5.000000,12.618075,\Rx:=0.000000,\Ry:=-5.366573),vel1,zoneval,Extruder\WObj:=Workobject_1;
MoveL RelTool (p1,25.500000,5.000000,11.328519,\Rx:=0.000000,\Ry:=-6.568275),vel1,zoneval,Extruder\WObj:=Workobject_1;
MoveL RelTool (p1,23.000000,5.000000,9.422774,\Rx:=0.000000,\Ry:=-9.481583),vel1,zoneval,Extruder\WObj:=Workobject_1;
MoveL RelTool (p1,20.500000,5.000000,6.707804,\Rx:=0.000000,\Ry:=-9.245066),vel1,zoneval,Extruder\WObj:=Workobject_1;
MoveL RelTool (p1,18.000000,5.000000,5.614048,\Rx:=0.000000,\Ry:=-3.081691),vel1,zoneval,Extruder\WObj:=Workobject_1;
MoveL RelTool (p1,15.500000,5.000000,5.500000,\Rx:=0.000000,\Ry:=-0.000000),vel1,zoneval,Extruder\WObj:=Workobject_1;
MoveL RelTool (p1,13.000000,5.000000,5.500000,\Rx:=0.000000,\Ry:=-0.000000),vel1,zoneval,Extruder\WObj:=Workobject_1;
MoveL RelTool (p1,10.500000,5.000000,5.500000,\Rx:=0.000000,\Ry:=-0.000000),vel1,zoneval,Extruder\WObj:=Workobject_1;
MoveL RelTool (p1,8.000000,5.000000,5.500000,\Rx:=0.000000,\Ry:=-0.000000),vel1,zoneval,Extruder\WObj:=Workobject_1;
MoveL RelTool (p1,5.500000,5.000000,5.500000,\Rx:=0.000000,\Ry:=-0.000000),vel1,zoneval,Extruder\WObj:=Workobject_1;
MoveL RelTool (p1,3.000000,5.000000,5.500000,\Rx:=0.000000,\Ry:=-0.000000),vel1,zoneval,Extruder\WObj:=Workobject_1;
MoveL RelTool (p1,5.000000,4.500000,5.500000,\Rx:=0.000000,\Ry:=0.000000),vel1,zoneval,Extruder\WObj:=Workobject_1;
MoveL RelTool (p1,7.500000,4.500000,5.500000,\Rx:=0.000000,\Ry:=0.000000),vel1,zoneval,Extruder\WObj:=Workobject_1;
MoveL RelTool (p1,10.000000,4.500000,5.500000,\Rx:=0.000000,\Ry:=0.000000),vel1,zoneval,Extruder\WObj:=Workobject_1;
MoveL RelTool (p1,12.500000,4.500000,5.500000,\Rx:=0.000000,\Ry:=0.000000),vel1,zoneval,Extruder\WObj:=Workobject_1;
MoveL RelTool (p1,15.000000,4.500000,5.500000,\Rx:=0.000000,\Ry:=0.000000),vel1,zoneval,Extruder\WObj:=Workobject_1;
MoveL RelTool (p1,17.500000,4.500000,5.549338,\Rx:=0.000000,\Ry:=-1.027233),vel1,zoneval,Extruder\WObj:=Workobject_1;
MoveL RelTool (p1,20.000000,4.500000,6.390765,\Rx:=0.000000,\Ry:=-6.482955),vel1,zoneval,Extruder\WObj:=Workobject_1;
MoveL RelTool (p1,22.500000,4.500000,8.916208,\Rx:=0.000000,\Ry:=-11.282192),vel1,zoneval,Extruder\WObj:=Workobject_1;
MoveL RelTool (p1,25.000000,4.500000,11.015814,\Rx:=0.000000,\Ry:=-7.926142),vel1,zoneval,Extruder\WObj:=Workobject_1;
MoveL RelTool (p1,27.500000,4.500000,12.393895,\Rx:=0.000000,\Ry:=-5.366573),vel1,zoneval,Extruder\WObj:=Workobject_1;
MoveL RelTool (p1,30.000000,4.500000,13.409588,\Rx:=0.000000,\Ry:=-4.304408),vel1,zoneval,Extruder\WObj:=Workobject_1;
MoveL RelTool (p1,32.500000,4.500000,14.177969,\Rx:=0.000000,\Ry:=-3.310711),vel1,zoneval,Extruder\WObj:=Workobject_1;
MoveL RelTool (p1,35.000000,4.500000,14.745289,\Rx:=0.000000,\Ry:=-2.361471),vel1,zoneval,Extruder\WObj:=Workobject_1;
MoveL RelTool (p1,37.500000,4.500000,15.140411,\Rx:=0.000000,\Ry:=-1.473255),vel1,zoneval,Extruder\WObj:=Workobject_1;
MoveL RelTool (p1,40.000000,4.500000,15.385044,\Rx:=0.000000,\Ry:=-0.609665),vel1,zoneval,Extruder\WObj:=Workobject_1;
MoveL RelTool (p1,42.500000,4.500000,15.493202,\Rx:=0.000000,\Ry:=-0.313643),vel1,zoneval,Extruder\WObj:=Workobject_1;
MoveL RelTool (p1,45.000000,4.500000,15.441995,\Rx:=0.000000,\Ry:=0.600478),vel1,zoneval,Extruder\WObj:=Workobject_1;
MoveL RelTool (p1,47.500000,4.500000,15.253646,\Rx:=0.000000,\Ry:=0.957446),vel1,zoneval,Extruder\WObj:=Workobject_1;
MoveL RelTool (p1,50.000000,4.500000,14.902666,\Rx:=0.000000,\Ry:=1.838961),vel1,zoneval,Extruder\WObj:=Workobject_1;
MoveL RelTool (p1,52.500000,4.500000,14.391107,\Rx:=0.000000,\Ry:=2.777529),vel1,zoneval,Extruder\WObj:=Workobject_1;
MoveL RelTool (p1,55.000000,4.500000,13.693467,\Rx:=0.000000,\Ry:=3.765598),vel1,zoneval,Extruder\WObj:=Workobject_1;
MoveL RelTool (p1,57.500000,4.500000,12.769306,\Rx:=0.000000,\Ry:=4.809648),vel1,zoneval,Extruder\WObj:=Workobject_1;
MoveL RelTool (p1,60.000000,4.500000,11.535030,\Rx:=0.000000,\Ry:=6.353659),vel1,zoneval,Extruder\WObj:=Workobject_1;
MoveL RelTool (p1,62.500000,4.500000,9.740509,\Rx:=0.000000,\Ry:=8.756273),vel1,zoneval,Extruder\WObj:=Workobject_1;
MoveL RelTool (p1,65.000000,4.500000,7.002928,\Rx:=0.000000,\Ry:=9.759467),vel1,zoneval,Extruder\WObj:=Workobject_1;
MoveL RelTool (p1,67.500000,4.500000,5.696103,\Rx:=0.000000,\Ry:=3.252694),vel1,zoneval,Extruder\WObj:=Workobject_1;
MoveL RelTool (p1,70.000000,4.500000,5.500000,\Rx:=0.000000,\Ry:=0.000000),vel1,zoneval,Extruder\WObj:=Workobject_1;
MoveL RelTool (p1,72.500000,4.500000,5.500000,\Rx:=0.000000,\Ry:=0.000000),vel1,zoneval,Extruder\WObj:=Workobject_1;
MoveL RelTool (p1,75.000000,4.500000,5.500000,\Rx:=0.000000,\Ry:=0.000000),vel1,zoneval,Extruder\WObj:=Workobject_1;
MoveL RelTool (p1,77.500000,4.500000,5.500000,\Rx:=0.000000,\Ry:=0.000000),vel1,zoneval,Extruder\WObj:=Workobject_1;
MoveL RelTool (p1,80.000000,4.500000,5.500000,\Rx:=0.000000,\Ry:=0.000000),vel1,zoneval,Extruder\WObj:=Workobject_1;
MoveL RelTool (p1,82.500000,4.500000,5.500000,\Rx:=0.000000,\Ry:=0.000000),vel1,zoneval,Extruder\WObj:=Workobject_1;
MoveL RelTool (p1,80.500000,4.000000,5.500000,\Rx:=0.000000,\Ry:=-0.000000),vel1,zoneval,Extruder\WObj:=Workobject_1;
MoveL RelTool (p1,78.000000,4.000000,5.500000,\Rx:=0.000000,\Ry:=-0.000000),vel1,zoneval,Extruder\WObj:=Workobject_1;
MoveL RelTool (p1,75.500000,4.000000,5.500000,\Rx:=0.000000,\Ry:=-0.000000),vel1,zoneval,Extruder\WObj:=Workobject_1;
MoveL RelTool (p1,73.000000,4.000000,5.500000,\Rx:=0.000000,\Ry:=-0.000000),vel1,zoneval,Extruder\WObj:=Workobject_1;
MoveL RelTool (p1,70.500000,4.000000,5.500000,\Rx:=0.000000,\Ry:=-0.000000),vel1,zoneval,Extruder\WObj:=Workobject_1;
MoveL RelTool (p1,68.000000,4.000000,5.576212,\Rx:=0.000000,\Ry:=1.027235),vel1,zoneval,Extruder\WObj:=Workobject_1;
MoveL RelTool (p1,65.500000,4.000000,6.601352,\Rx:=0.000000,\Ry:=7.190651),vel1,zoneval,Extruder\WObj:=Workobject_1;
MoveL RelTool (p1,63.000000,4.000000,9.259802,\Rx:=0.000000,\Ry:=10.438096),vel1,zoneval,Extruder\WObj:=Workobject_1;
MoveL RelTool (p1,60.500000,4.000000,11.213438,\Rx:=0.000000,\Ry:=7.277441),vel1,zoneval,Extruder\WObj:=Workobject_1;
MoveL RelTool (p1,58.000000,4.000000,12.567025,\Rx:=0.000000,\Ry:=5.967579),vel1,zoneval,Extruder\WObj:=Workobject_1;
MoveL RelTool (p1,55.500000,4.000000,13.541124,\Rx:=0.000000,\Ry:=4.323199),vel1,zoneval,Extruder\WObj:=Workobject_1;
MoveL RelTool (p1,53.000000,4.000000,14.280270,\Rx:=0.000000,\Ry:=3.233363),vel1,zoneval,Extruder\WObj:=Workobject_1;
MoveL RelTool (p1,50.500000,4.000000,14.829944,\Rx:=0.000000,\Ry:=2.667808),vel1,zoneval,Extruder\WObj:=Workobject_1;
MoveL RelTool (p1,48.000000,4.000000,15.193555,\Rx:=0.000000,\Ry:=1.838961),vel1,zoneval,Extruder\WObj:=Workobject_1;
MoveL RelTool (p1,45.500000,4.000000,15.404325,\Rx:=0.000000,\Ry:=0.957446),vel1,zoneval,Extruder\WObj:=Workobject_1;
MoveL RelTool (p1,43.000000,4.000000,15.486300,\Rx:=0.000000,\Ry:=0.175753),vel1,zoneval,Extruder\WObj:=Workobject_1;
MoveL RelTool (p1,40.500000,4.000000,15.409004,\Rx:=0.000000,\Ry:=-0.609665),vel1,zoneval,Extruder\WObj:=Workobject_1;
MoveL RelTool (p1,38.000000,4.000000,15.198525,\Rx:=0.000000,\Ry:=-1.473255),vel1,zoneval,Extruder\WObj:=Workobject_1;
MoveL RelTool (p1,35.500000,4.000000,14.839102,\Rx:=0.000000,\Ry:=-2.361471),vel1,zoneval,Extruder\WObj:=Workobject_1;
MoveL RelTool (p1,33.000000,4.000000,14.310992,\Rx:=0.000000,\Ry:=-3.310711),vel1,zoneval,Extruder\WObj:=Workobject_1;
MoveL RelTool (p1,30.500000,4.000000,13.585370,\Rx:=0.000000,\Ry:=-4.304408),vel1,zoneval,Extruder\WObj:=Workobject_1;
MoveL RelTool (p1,28.000000,4.000000,12.618075,\Rx:=0.000000,\Ry:=-5.366573),vel1,zoneval,Extruder\WObj:=Workobject_1;
MoveL RelTool (p1,25.500000,4.000000,11.328519,\Rx:=0.000000,\Ry:=-6.568275),vel1,zoneval,Extruder\WObj:=Workobject_1;
MoveL RelTool (p1,23.000000,4.000000,9.422774,\Rx:=0.000000,\Ry:=-9.481583),vel1,zoneval,Extruder\WObj:=Workobject_1;
MoveL RelTool (p1,20.500000,4.000000,6.707804,\Rx:=0.000000,\Ry:=-9.245066),vel1,zoneval,Extruder\WObj:=Workobject_1;
MoveL RelTool (p1,18.000000,4.000000,5.614048,\Rx:=0.000000,\Ry:=-3.081691),vel1,zoneval,Extruder\WObj:=Workobject_1;
MoveL RelTool (p1,15.500000,4.000000,5.500000,\Rx:=0.000000,\Ry:=-0.000000),vel1,zoneval,Extruder\WObj:=Workobject_1;
MoveL RelTool (p1,13.000000,4.000000,5.500000,\Rx:=0.000000,\Ry:=-0.000000),vel1,zoneval,Extruder\WObj:=Workobject_1;
MoveL RelTool (p1,10.500000,4.000000,5.500000,\Rx:=0.000000,\Ry:=-0.000000),vel1,zoneval,Extruder\WObj:=Workobject_1;
MoveL RelTool (p1,8.000000,4.000000,5.500000,\Rx:=0.000000,\Ry:=-0.000000),vel1,zoneval,Extruder\WObj:=Workobject_1;
MoveL RelTool (p1,5.500000,4.000000,5.500000,\Rx:=0.000000,\Ry:=-0.000000),vel1,zoneval,Extruder\WObj:=Workobject_1;
MoveL RelTool (p1,3.000000,4.000000,5.500000,\Rx:=0.000000,\Ry:=-0.000000),vel1,zoneval,Extruder\WObj:=Workobject_1;
MoveL RelTool (p1,5.000000,3.500000,5.500000,\Rx:=0.000000,\Ry:=0.000000),vel1,zoneval,Extruder\WObj:=Workobject_1;
MoveL RelTool (p1,7.500000,3.500000,5.500000,\Rx:=0.000000,\Ry:=0.000000),vel1,zoneval,Extruder\WObj:=Workobject_1;
MoveL RelTool (p1,10.000000,3.500000,5.500000,\Rx:=0.000000,\Ry:=0.000000),vel1,zoneval,Extruder\WObj:=Workobject_1;
MoveL RelTool (p1,12.500000,3.500000,5.500000,\Rx:=0.000000,\Ry:=0.000000),vel1,zoneval,Extruder\WObj:=Workobject_1;
MoveL RelTool (p1,15.000000,3.500000,5.500000,\Rx:=0.000000,\Ry:=0.000000),vel1,zoneval,Extruder\WObj:=Workobject_1;
MoveL RelTool (p1,17.500000,3.500000,5.549338,\Rx:=0.000000,\Ry:=-1.027233),vel1,zoneval,Extruder\WObj:=Workobject_1;
MoveL RelTool (p1,20.000000,3.500000,6.390765,\Rx:=0.000000,\Ry:=-6.482955),vel1,zoneval,Extruder\WObj:=Workobject_1;
MoveL RelTool (p1,22.500000,3.500000,8.916208,\Rx:=0.000000,\Ry:=-11.282192),vel1,zoneval,Extruder\WObj:=Workobject_1;
MoveL RelTool (p1,25.000000,3.500000,11.015814,\Rx:=0.000000,\Ry:=-7.926142),vel1,zoneval,Extruder\WObj:=Workobject_1;
MoveL RelTool (p1,27.500000,3.500000,12.393895,\Rx:=0.000000,\Ry:=-5.366573),vel1,zoneval,Extruder\WObj:=Workobject_1;
MoveL RelTool (p1,30.000000,3.500000,13.409588,\Rx:=0.000000,\Ry:=-4.304408),vel1,zoneval,Extruder\WObj:=Workobject_1;
MoveL RelTool (p1,32.500000,3.500000,14.177969,\Rx:=0.000000,\Ry:=-3.310711),vel1,zoneval,Extruder\WObj:=Workobject_1;
MoveL RelTool (p1,35.000000,3.500000,14.745289,\Rx:=0.000000,\Ry:=-2.361471),vel1,zoneval,Extruder\WObj:=Workobject_1;
MoveL RelTool (p1,37.500000,3.500000,15.140411,\Rx:=0.000000,\Ry:=-1.473255),vel1,zoneval,Extruder\WObj:=Workobject_1;
MoveL RelTool (p1,40.000000,3.500000,15.385044,\Rx:=0.000000,\Ry:=-0.609665),vel1,zoneval,Extruder\WObj:=Workobject_1;
MoveL RelTool (p1,42.500000,3.500000,15.493202,\Rx:=0.000000,\Ry:=-0.313643),vel1,zoneval,Extruder\WObj:=Workobject_1;
MoveL RelTool (p1,45.000000,3.500000,15.441995,\Rx:=0.000000,\Ry:=0.600478),vel1,zoneval,Extruder\WObj:=Workobject_1;
MoveL RelTool (p1,47.500000,3.500000,15.253646,\Rx:=0.000000,\Ry:=0.957446),vel1,zoneval,Extruder\WObj:=Workobject_1;
MoveL RelTool (p1,50.000000,3.500000,14.902666,\Rx:=0.000000,\Ry:=1.838961),vel1,zoneval,Extruder\WObj:=Workobject_1;
MoveL RelTool (p1,52.500000,3.500000,14.391107,\Rx:=0.000000,\Ry:=2.777529),vel1,zoneval,Extruder\WObj:=Workobject_1;
MoveL RelTool (p1,55.000000,3.500000,13.693467,\Rx:=0.000000,\Ry:=3.765598),vel1,zoneval,Extruder\WObj:=Workobject_1;
MoveL RelTool (p1,57.500000,3.500000,12.769306,\Rx:=0.000000,\Ry:=4.809648),vel1,zoneval,Extruder\WObj:=Workobject_1;
MoveL RelTool (p1,60.000000,3.500000,11.535030,\Rx:=0.000000,\Ry:=6.353659),vel1,zoneval,Extruder\WObj:=Workobject_1;
MoveL RelTool (p1,62.500000,3.500000,9.740509,\Rx:=0.000000,\Ry:=8.756273),vel1,zoneval,Extruder\WObj:=Workobject_1;
MoveL RelTool (p1,65.000000,3.500000,7.002928,\Rx:=0.000000,\Ry:=9.759467),vel1,zoneval,Extruder\WObj:=Workobject_1;
MoveL RelTool (p1,67.500000,3.500000,5.696103,\Rx:=0.000000,\Ry:=3.252694),vel1,zoneval,Extruder\WObj:=Workobject_1;
MoveL RelTool (p1,70.000000,3.500000,5.500000,\Rx:=0.000000,\Ry:=0.000000),vel1,zoneval,Extruder\WObj:=Workobject_1;
MoveL RelTool (p1,72.500000,3.500000,5.500000,\Rx:=0.000000,\Ry:=0.000000),vel1,zoneval,Extruder\WObj:=Workobject_1;
MoveL RelTool (p1,75.000000,3.500000,5.500000,\Rx:=0.000000,\Ry:=0.000000),vel1,zoneval,Extruder\WObj:=Workobject_1;
MoveL RelTool (p1,77.500000,3.500000,5.500000,\Rx:=0.000000,\Ry:=0.000000),vel1,zoneval,Extruder\WObj:=Workobject_1;
MoveL RelTool (p1,80.000000,3.500000,5.500000,\Rx:=0.000000,\Ry:=0.000000),vel1,zoneval,Extruder\WObj:=Workobject_1;
MoveL RelTool (p1,82.500000,3.500000,5.500000,\Rx:=0.000000,\Ry:=0.000000),vel1,zoneval,Extruder\WObj:=Workobject_1;
MoveL RelTool (p1,80.500000,3.000000,5.500000,\Rx:=0.000000,\Ry:=-0.000000),vel1,zoneval,Extruder\WObj:=Workobject_1;
MoveL RelTool (p1,78.000000,3.000000,5.500000,\Rx:=0.000000,\Ry:=-0.000000),vel1,zoneval,Extruder\WObj:=Workobject_1;
MoveL RelTool (p1,75.500000,3.000000,5.500000,\Rx:=0.000000,\Ry:=-0.000000),vel1,zoneval,Extruder\WObj:=Workobject_1;
